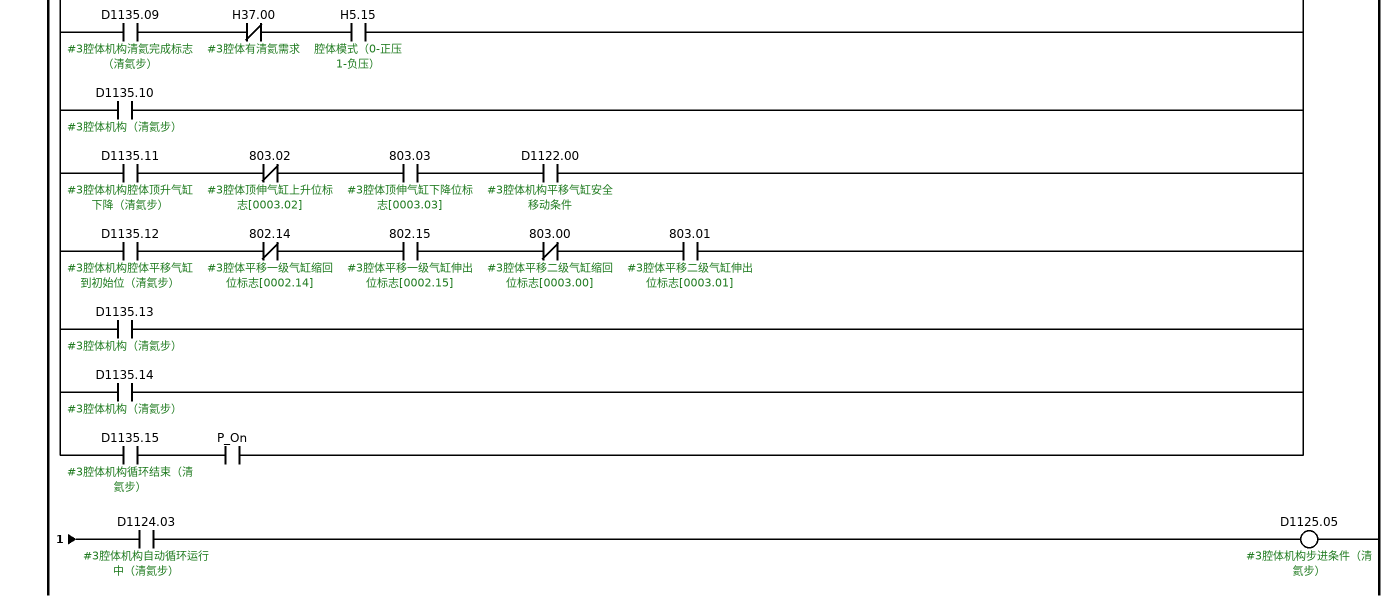
; [picture p312: 氦检机构 / 氦检腔3自动, rungs 23-23]
; rung 23
LD D1134.00  ; #3腔体机构自动开始（清氦步）
AND T1576  ; #3腔体机构开始运行延时（清氦步）
LD D1134.01  ; #3腔体机构平移气缸到氦检位/数据初始化（清氦步）
ANDNOT 802.14  ; #3腔体平移一级气缸缩回位标志[0002.14]
AND 802.15  ; #3腔体平移一级气缸伸出位标志[0002.15]
AND 803.00  ; #3腔体平移二级气缸缩回位标志[0003.00]
ANDNOT 803.01  ; #3腔体平移二级气缸伸出位标志[0003.01]
AND T2140  ; #3-1数据初始化延时（清氦）
ORLD
LD D1134.02  ; #3腔体机构腔体顶升气缸上升（清氦步）
AND 803.02  ; #3腔体顶伸气缸上升位标志[0003.02]
ANDNOT 803.03  ; #3腔体顶伸气缸下降位标志[0003.03]
ORLD
LD D1134.03  ; #3腔体机构氦检仪真空阀关闭（清氦步）
AND 820.11  ; 氦检仪真空阀关到位标志
ORLD
LD D1134.04  ; #3腔体机构正压开腔体阀/负压关腔体阀/氦检阀打开  // 负压模式下，复测前的清氦不允许抽电池
LDNOT H5.15  ; 腔体模式（0-正压 1-负压）
ORNOT D1127.01  ; #3腔体机构清氦需求判定（自动步）
LD 822.04  ; #3-1腔体阀开到位标志
AND 822.06  ; #3-2腔体阀开到位标志
LD D1130.11  ; #3腔体机构关闭#3-1腔体阀/清氦判定（自动单检步）
AND 822.04  ; #3-1腔体阀开到位标志
ORLD
LD D1131.07  ; #3腔体机构清氦需求判定（自动单检步）
AND 822.06  ; #3-2腔体阀开到位标志
ORLD
ANDLD
LD H5.15  ; 腔体模式（0-正压 1-负压）
AND D1127.01  ; #3腔体机构清氦需求判定（自动步）
AND 822.05  ; #3-1腔体阀关到位标志
AND 822.07  ; #3-2腔体阀关到位标志
ORLD
ANDLD
AND D1122.15  ; #3腔体机构腔体抽气阀打开允许
AND D1122.14  ; #3腔体氦检阀打开允许条件
AND 803.04  ; #3腔体氦检阀开到位标志[0003.04]
LD W380.15  ; 氦检仪漏率低于设定值（稳态）
OR H5.02  ; 氦检仪屏蔽
ANDLD
ORLD
OR D1134.05  ; #3腔体机构（清氦步）
LD D1134.06  ; #3腔体机构腔体抽气阀打开/电池抽气阀打开（清氦步）
LD T2100  ; #3-1腔体抽真空阈值到达延时（测试）
OR T2108  ; #3-1腔体抽残气时间上限到达延时（测试）
ANDLD
LD 824.04  ; #3-1电池抽真空阀开到位标志
AND T2120  ; #3-1电池抽真空阈值到达延时（测试）
OR T2121  ; #3-1电池抽真空时间上限到达延时（测试）
LD 824.06  ; #3-2电池抽真空阀开到位标志
AND T2420  ; #3-2电池抽真空阈值到达延时（测试）
OR T2421  ; #3-2电池抽真空时间上限到达延时（测试）
ANDLD
OR H5.15  ; 腔体模式（0-正压 1-负压）
OR H5.10  ; 空跑程序
ANDLD
ORLD
LD D1134.07  ; #3腔体机构腔体抽气阀关闭/电池抽气阀关闭（清氦步）
AND 822.03  ; #3腔体抽真空阀关到位标志
AND 824.05  ; #3-1电池抽真空阀关到位标志
AND 824.07  ; #3-2电池抽真空阀关到位标志
ORLD
OR D1134.08  ; #3腔体机构（清氦步）
LD D1134.09  ; #3腔体机构氦检清洁阀打开/电池破真空阀打开（清氦步）
AND T2141  ; #3-1清氦注氮时长（清氦）
LD T2122  ; #3-1电池破真空阈值到达延时（测试）
OR T2123  ; #3-1电池破真空时间上限到达延时（测试）
ANDLD
LD T2422  ; #3-2电池破真空阈值到达延时（测试）
OR T2423  ; #3-2电池破真空时间上限到达延时（测试）
ANDLD
ORLD
LD D1134.10  ; #3腔体机构氦检清洁阀关闭/电池破真空阀关闭（清氦步）
AND 820.13  ; 复检清洁阀关到位标志
AND 824.13  ; #3-1电池破真空阀关到位标志
AND 824.15  ; #3-2电池破真空阀关到位标志
ORLD
OR D1134.11  ; #3腔体机构（清氦步）
LD D1134.12  ; #3腔体机构清氦次数判定（清氦步）
AND>=(325) D472 D124  ; #3-1腔体管路清氦计数, 腔体测试设定清氦次数（次_UInt）
ORLD
OR D1134.13  ; #3腔体机构（清氦步）
LD D1134.14  ; #3腔体机构腔体抽气阀打开/电池抽气阀打开（清氦步）
AND 803.04  ; #3腔体氦检阀开到位标志[0003.04]
AND T2100  ; #3-1腔体抽真空阈值到达延时（测试）
LD 824.04  ; #3-1电池抽真空阀开到位标志
AND T2120  ; #3-1电池抽真空阈值到达延时（测试）
AND 824.06  ; #3-2电池抽真空阀开到位标志
AND T2420  ; #3-2电池抽真空阈值到达延时（测试）
OR H5.15  ; 腔体模式（0-正压 1-负压）
OR H5.10  ; 空跑程序
ANDLD
ORLD
LD D1134.15  ; #3腔体机构关闭电池抽气阀（清氦步）
AND 824.05  ; #3-1电池抽真空阀关到位标志
AND 824.07  ; #3-2电池抽真空阀关到位标志
ORLD
LD D1135.00  ; #3腔体机构腔体氦检阀仪真空阀打开/延时关腔体抽气阀（清氦步）
AND 803.04  ; #3腔体氦检阀开到位标志[0003.04]
AND 820.10  ; 氦检仪真空阀开到位标志
AND T2106  ; #3-1腔体氦检数据取值判定延时（测试）
ORLD
OR D1135.01  ; #3腔体机构（清氦步）
LD D1135.02  ; #3腔体机构腔体氦检阀关闭（清氦步）
AND 803.05  ; #3腔体氦检阀关到位标志[0003.05]
ORLD
LD D1135.03  ; #3腔体机构腔体抽气阀关闭/电池抽气阀关闭（清氦步）
AND 824.05  ; #3-1电池抽真空阀关到位标志
AND 824.07  ; #3-2电池抽真空阀关到位标志
AND 822.03  ; #3腔体抽真空阀关到位标志
ORLD
LD D1135.04  ; #3腔体机构是否需要重新清氦判定（清氦步）
ANDNOT H37.10  ; #3-1腔体清氦失败，重新进行清氦流程  // 清氦失败，重新进行清氦
ORLD
OR D1135.05  ; #3腔体机构（清氦步）
LD D1135.06  ; #3腔体机构开腔体破真空阀/开电池破真空阀/开腔体阀（清氦步）
AND T2102  ; #3-1腔体破真空阈值到达延时（测试）
AND T2122  ; #3-1电池破真空阈值到达延时（测试）
AND T2422  ; #3-2电池破真空阈值到达延时（测试）
ORLD
LD D1135.07  ; #3腔体机构关腔体破真空阀/关电池破真空阀（清氦步）
AND 822.09  ; #3腔体破真空阀关到位标志
AND 824.13  ; #3-1电池破真空阀关到位标志
AND 824.15  ; #3-2电池破真空阀关到位标志
ORLD
OR D1135.08  ; #3腔体机构（清氦步）
LD D1135.09  ; #3腔体机构清氦完成标志（清氦步）  // 正压腔体是待料清氦，需跳转回测试步序
ANDNOT H37.00  ; #3腔体有清氦需求
AND H5.15  ; 腔体模式（0-正压 1-负压）
ORLD
OR D1135.10  ; #3腔体机构（清氦步）
LD D1135.11  ; #3腔体机构腔体顶升气缸下降（清氦步）
ANDNOT 803.02  ; #3腔体顶伸气缸上升位标志[0003.02]
AND 803.03  ; #3腔体顶伸气缸下降位标志[0003.03]
AND D1122.00  ; #3腔体机构平移气缸安全移动条件
ORLD
LD D1135.12  ; #3腔体机构腔体平移气缸到初始位（清氦步）
ANDNOT 802.14  ; #3腔体平移一级气缸缩回位标志[0002.14]
AND 802.15  ; #3腔体平移一级气缸伸出位标志[0002.15]
ANDNOT 803.00  ; #3腔体平移二级气缸缩回位标志[0003.00]
AND 803.01  ; #3腔体平移二级气缸伸出位标志[0003.01]
ORLD
OR D1135.13  ; #3腔体机构（清氦步）
OR D1135.14  ; #3腔体机构（清氦步）
LD D1135.15  ; #3腔体机构循环结束（清氦步）
AND P_On
ORLD
AND D1124.03  ; #3腔体机构自动循环运行中（清氦步）
OUT D1125.05  ; #3腔体机构步进条件（清氦步）

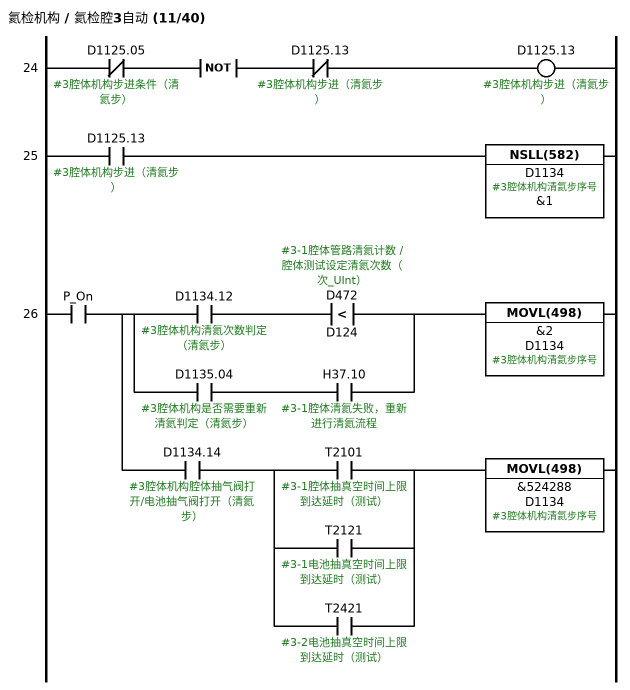
; rung 24
LDNOT D1125.05  ; #3腔体机构步进条件（清氦步）
NOT(520)
ANDNOT D1125.13  ; #3腔体机构步进（清氦步）
OUT D1125.13  ; #3腔体机构步进（清氦步）
; rung 25
LD D1125.13  ; #3腔体机构步进（清氦步）
NSLL(582) D1134 &1  ; #3腔体机构清氦步序号
; rung 26
LD P_On
OUT TR0
LD D1134.12  ; #3腔体机构清氦次数判定（清氦步）
AND<(310) D472 D124  ; #3-1腔体管路清氦计数, 腔体测试设定清氦次数（次_UInt）
LD D1135.04  ; #3腔体机构是否需要重新清氦判定（清氦步）
AND H37.10  ; #3-1腔体清氦失败，重新进行清氦流程  // 清氦失败，重新进行清氦
ORLD
ANDLD
MOVL(498) &2 D1134  ; #3腔体机构清氦步序号
LD TR0
AND D1134.14  ; #3腔体机构腔体抽气阀打开/电池抽气阀打开（清氦步）
LD T2101  ; #3-1腔体抽真空时间上限到达延时（测试）
OR T2121  ; #3-1电池抽真空时间上限到达延时（测试）
OR T2421  ; #3-2电池抽真空时间上限到达延时（测试）
ANDLD
MOVL(498) &524288 D1134  ; #3腔体机构清氦步序号  // 清氦过程腔体或电池抽气上限达到，均直接判定清氦完成，不进入氦检步序（跳转至D1075.03）

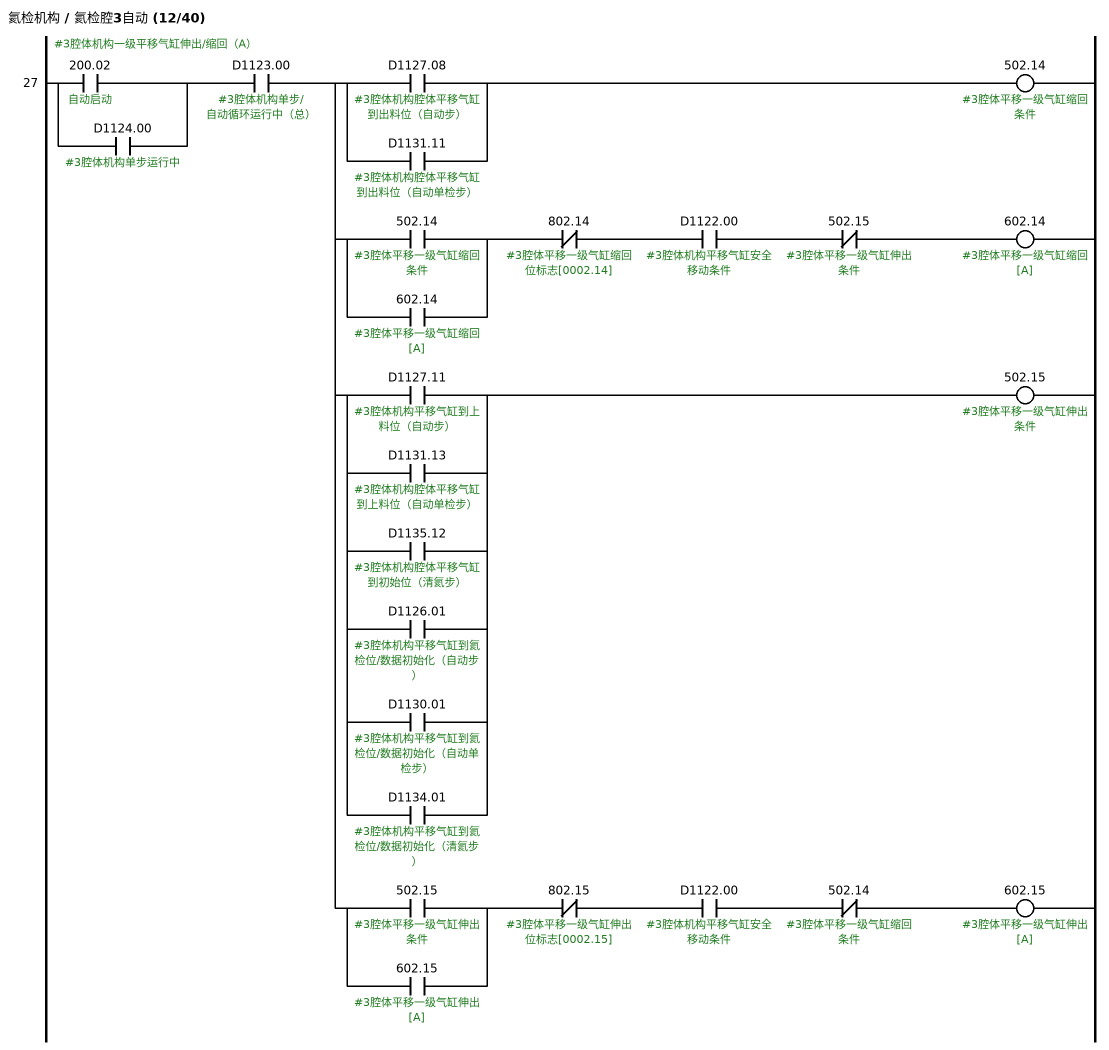
; rung 27: #3腔体机构一级平移气缸伸出/缩回（A）
LD 200.02  ; 自动启动
OR D1124.00  ; #3腔体机构单步运行中
AND D1123.00  ; #3腔体机构单步/自动循环运行中（总）
OUT TR0
LD D1127.08  ; #3腔体机构腔体平移气缸到出料位（自动步）
OR D1131.11  ; #3腔体机构腔体平移气缸到出料位（自动单检步）
ANDLD
OUT 502.14  ; #3腔体平移一级气缸缩回条件
LD TR0
LD 502.14  ; #3腔体平移一级气缸缩回条件
OR 602.14  ; #3腔体平移一级气缸缩回[A]
ANDLD
ANDNOT 802.14  ; #3腔体平移一级气缸缩回位标志[0002.14]
AND D1122.00  ; #3腔体机构平移气缸安全移动条件
ANDNOT 502.15  ; #3腔体平移一级气缸伸出条件
OUT 602.14  ; #3腔体平移一级气缸缩回[A]
LD TR0
LD D1127.11  ; #3腔体机构平移气缸到上料位（自动步）
OR D1131.13  ; #3腔体机构腔体平移气缸到上料位（自动单检步）
OR D1135.12  ; #3腔体机构腔体平移气缸到初始位（清氦步）
OR D1126.01  ; #3腔体机构平移气缸到氦检位/数据初始化（自动步）
OR D1130.01  ; #3腔体机构平移气缸到氦检位/数据初始化（自动单检步）
OR D1134.01  ; #3腔体机构平移气缸到氦检位/数据初始化（清氦步）
ANDLD
OUT 502.15  ; #3腔体平移一级气缸伸出条件
LD TR0
LD 502.15  ; #3腔体平移一级气缸伸出条件
OR 602.15  ; #3腔体平移一级气缸伸出[A]
ANDLD
ANDNOT 802.15  ; #3腔体平移一级气缸伸出位标志[0002.15]
AND D1122.00  ; #3腔体机构平移气缸安全移动条件
ANDNOT 502.14  ; #3腔体平移一级气缸缩回条件
OUT 602.15  ; #3腔体平移一级气缸伸出[A]

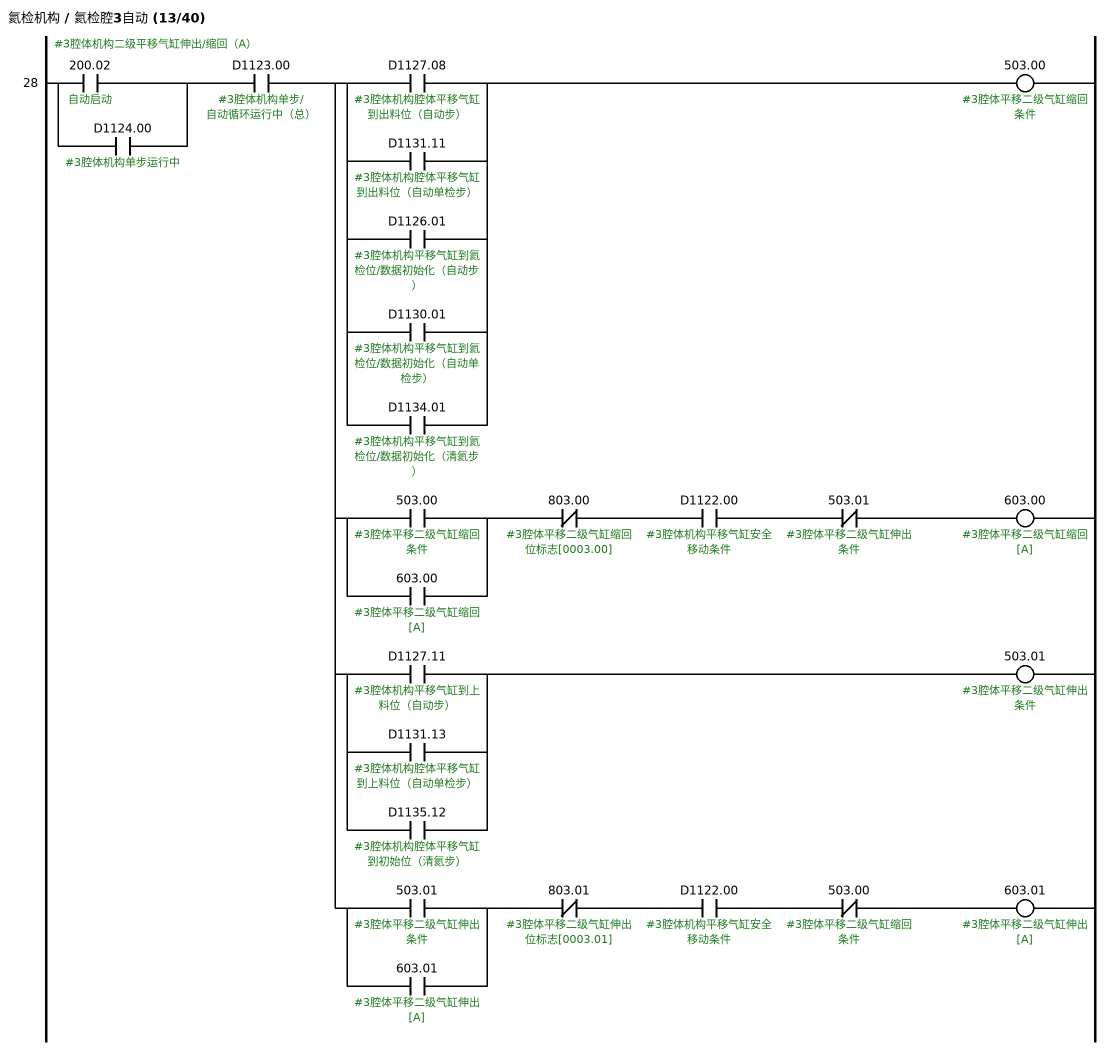
; rung 28: #3腔体机构二级平移气缸伸出/缩回（A）
LD 200.02  ; 自动启动
OR D1124.00  ; #3腔体机构单步运行中
AND D1123.00  ; #3腔体机构单步/自动循环运行中（总）
OUT TR0
LD D1127.08  ; #3腔体机构腔体平移气缸到出料位（自动步）
OR D1131.11  ; #3腔体机构腔体平移气缸到出料位（自动单检步）
OR D1126.01  ; #3腔体机构平移气缸到氦检位/数据初始化（自动步）
OR D1130.01  ; #3腔体机构平移气缸到氦检位/数据初始化（自动单检步）
OR D1134.01  ; #3腔体机构平移气缸到氦检位/数据初始化（清氦步）
ANDLD
OUT 503.00  ; #3腔体平移二级气缸缩回条件
LD TR0
LD 503.00  ; #3腔体平移二级气缸缩回条件
OR 603.00  ; #3腔体平移二级气缸缩回[A]
ANDLD
ANDNOT 803.00  ; #3腔体平移二级气缸缩回位标志[0003.00]
AND D1122.00  ; #3腔体机构平移气缸安全移动条件
ANDNOT 503.01  ; #3腔体平移二级气缸伸出条件
OUT 603.00  ; #3腔体平移二级气缸缩回[A]
LD TR0
LD D1127.11  ; #3腔体机构平移气缸到上料位（自动步）
OR D1131.13  ; #3腔体机构腔体平移气缸到上料位（自动单检步）
OR D1135.12  ; #3腔体机构腔体平移气缸到初始位（清氦步）
ANDLD
OUT 503.01  ; #3腔体平移二级气缸伸出条件
LD TR0
LD 503.01  ; #3腔体平移二级气缸伸出条件
OR 603.01  ; #3腔体平移二级气缸伸出[A]
ANDLD
ANDNOT 803.01  ; #3腔体平移二级气缸伸出位标志[0003.01]
AND D1122.00  ; #3腔体机构平移气缸安全移动条件
ANDNOT 503.00  ; #3腔体平移二级气缸缩回条件
OUT 603.01  ; #3腔体平移二级气缸伸出[A]

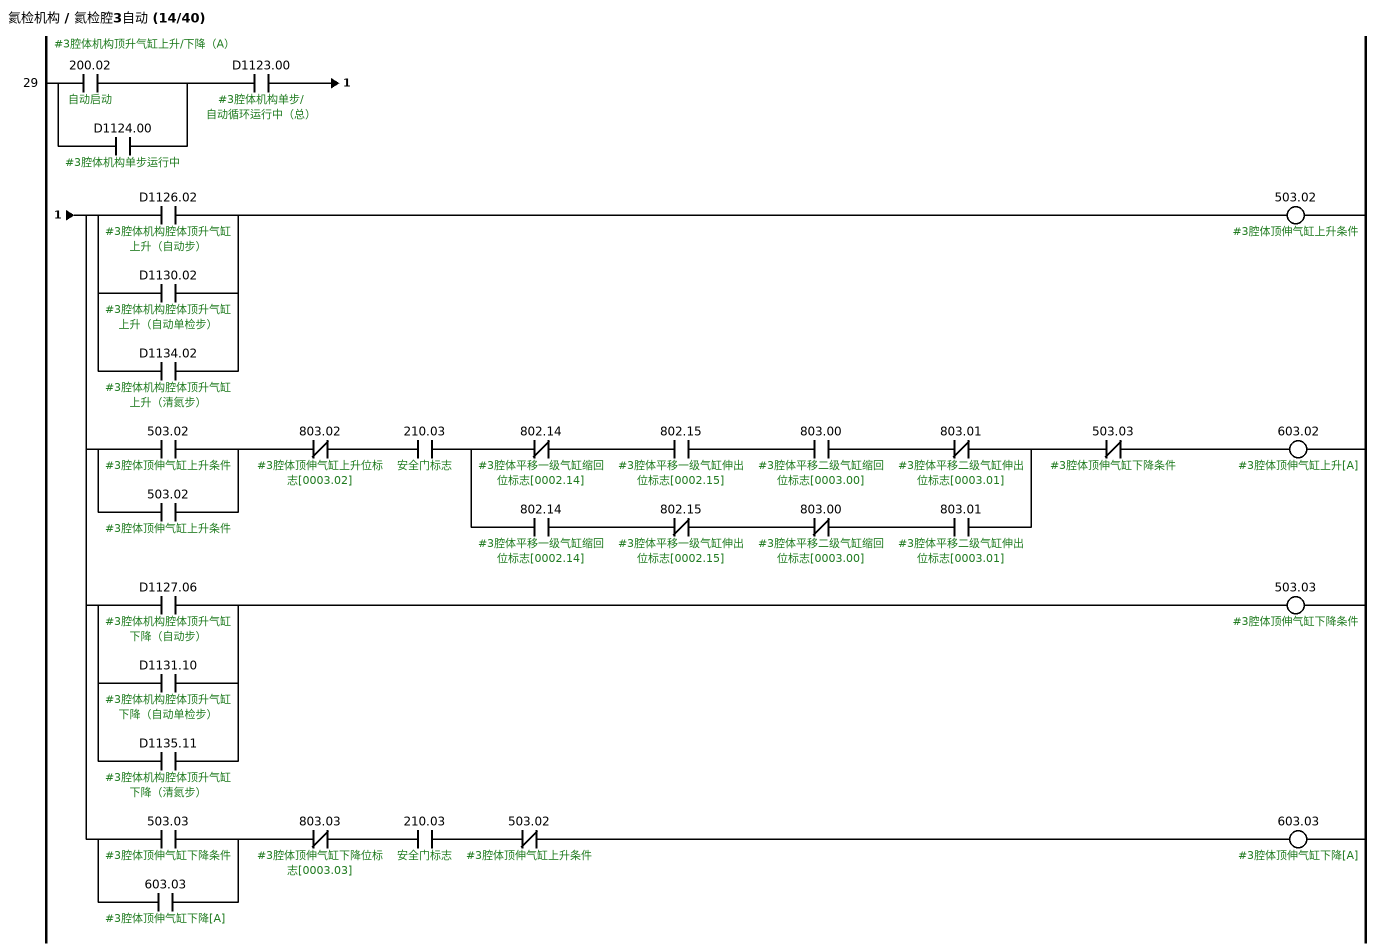
; rung 29: #3腔体机构顶升气缸上升/下降（A）
LD 200.02  ; 自动启动
OR D1124.00  ; #3腔体机构单步运行中
AND D1123.00  ; #3腔体机构单步/自动循环运行中（总）
OUT TR0
LD D1126.02  ; #3腔体机构腔体顶升气缸上升（自动步）
OR D1130.02  ; #3腔体机构腔体顶升气缸上升（自动单检步）
OR D1134.02  ; #3腔体机构腔体顶升气缸上升（清氦步）
ANDLD
OUT 503.02  ; #3腔体顶伸气缸上升条件
LD TR0
LD 503.02  ; #3腔体顶伸气缸上升条件
OR 503.02  ; #3腔体顶伸气缸上升条件
ANDLD
ANDNOT 803.02  ; #3腔体顶伸气缸上升位标志[0003.02]
AND 210.03  ; 安全门标志
LDNOT 802.14  ; #3腔体平移一级气缸缩回位标志[0002.14]
AND 802.15  ; #3腔体平移一级气缸伸出位标志[0002.15]
AND 803.00  ; #3腔体平移二级气缸缩回位标志[0003.00]
ANDNOT 803.01  ; #3腔体平移二级气缸伸出位标志[0003.01]
LD 802.14  ; #3腔体平移一级气缸缩回位标志[0002.14]
ANDNOT 802.15  ; #3腔体平移一级气缸伸出位标志[0002.15]
ANDNOT 803.00  ; #3腔体平移二级气缸缩回位标志[0003.00]
AND 803.01  ; #3腔体平移二级气缸伸出位标志[0003.01]
ORLD
ANDLD
ANDNOT 503.03  ; #3腔体顶伸气缸下降条件
OUT 603.02  ; #3腔体顶伸气缸上升[A]
LD TR0
LD D1127.06  ; #3腔体机构腔体顶升气缸下降（自动步）
OR D1131.10  ; #3腔体机构腔体顶升气缸下降（自动单检步）
OR D1135.11  ; #3腔体机构腔体顶升气缸下降（清氦步）
ANDLD
OUT 503.03  ; #3腔体顶伸气缸下降条件
LD TR0
LD 503.03  ; #3腔体顶伸气缸下降条件
OR 603.03  ; #3腔体顶伸气缸下降[A]
ANDLD
ANDNOT 803.03  ; #3腔体顶伸气缸下降位标志[0003.03]
AND 210.03  ; 安全门标志
ANDNOT 503.02  ; #3腔体顶伸气缸上升条件
OUT 603.03  ; #3腔体顶伸气缸下降[A]

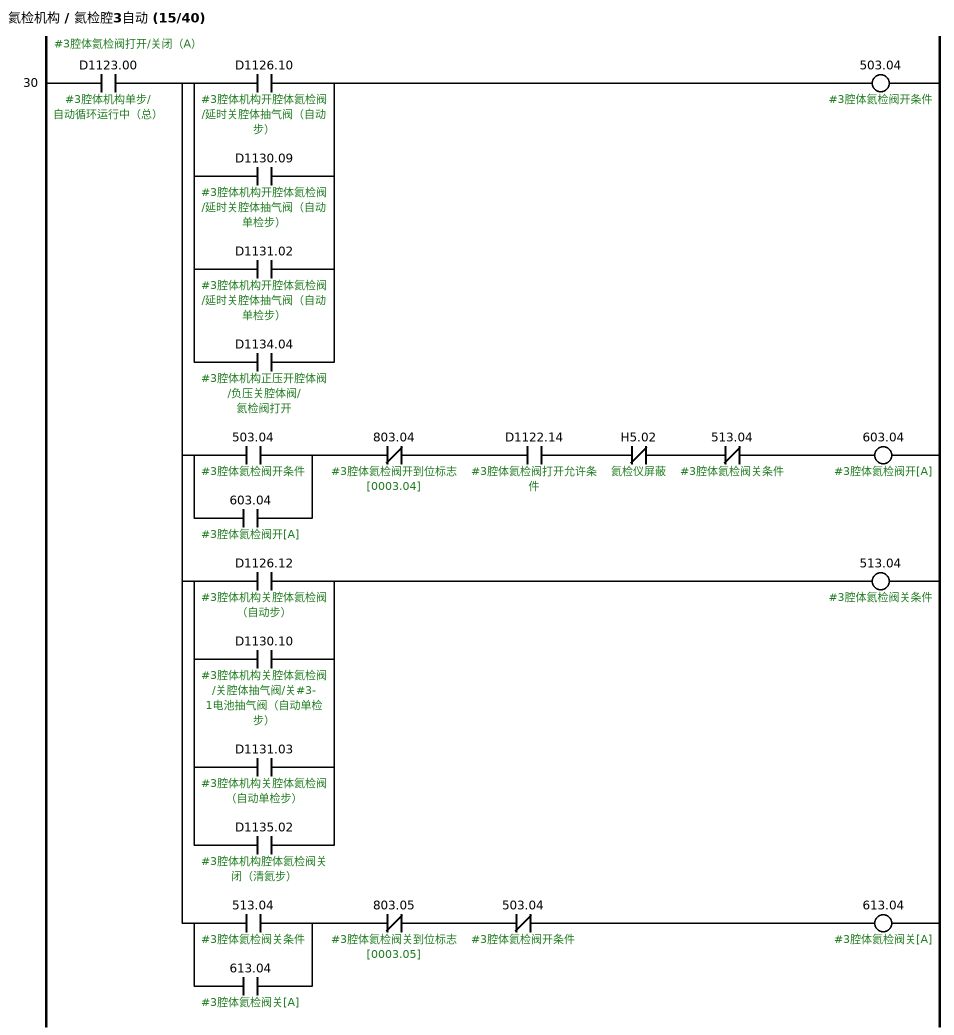
; rung 30: #3腔体氦检阀打开/关闭（A）
LD D1123.00  ; #3腔体机构单步/自动循环运行中（总）
OUT TR0
LD D1126.10  ; #3腔体机构开腔体氦检阀/延时关腔体抽气阀（自动步）
OR D1130.09  ; #3腔体机构开腔体氦检阀/延时关腔体抽气阀（自动单检步）
OR D1131.02  ; #3腔体机构开腔体氦检阀/延时关腔体抽气阀（自动单检步）
OR D1134.04  ; #3腔体机构正压开腔体阀/负压关腔体阀/氦检阀打开
ANDLD
OUT 503.04  ; #3腔体氦检阀开条件
LD TR0
LD 503.04  ; #3腔体氦检阀开条件
OR 603.04  ; #3腔体氦检阀开[A]
ANDLD
ANDNOT 803.04  ; #3腔体氦检阀开到位标志[0003.04]
AND D1122.14  ; #3腔体氦检阀打开允许条件
ANDNOT H5.02  ; 氦检仪屏蔽
ANDNOT 513.04  ; #3腔体氦检阀关条件
OUT 603.04  ; #3腔体氦检阀开[A]
LD TR0
LD D1126.12  ; #3腔体机构关腔体氦检阀（自动步）
OR D1130.10  ; #3腔体机构关腔体氦检阀/关腔体抽气阀/关#3-1电池抽气阀（自动单检步）
OR D1131.03  ; #3腔体机构关腔体氦检阀（自动单检步）
OR D1135.02  ; #3腔体机构腔体氦检阀关闭（清氦步）
ANDLD
OUT 513.04  ; #3腔体氦检阀关条件
LD TR0
LD 513.04  ; #3腔体氦检阀关条件
OR 613.04  ; #3腔体氦检阀关[A]
ANDLD
ANDNOT 803.05  ; #3腔体氦检阀关到位标志[0003.05]
ANDNOT 503.04  ; #3腔体氦检阀开条件
OUT 613.04  ; #3腔体氦检阀关[A]

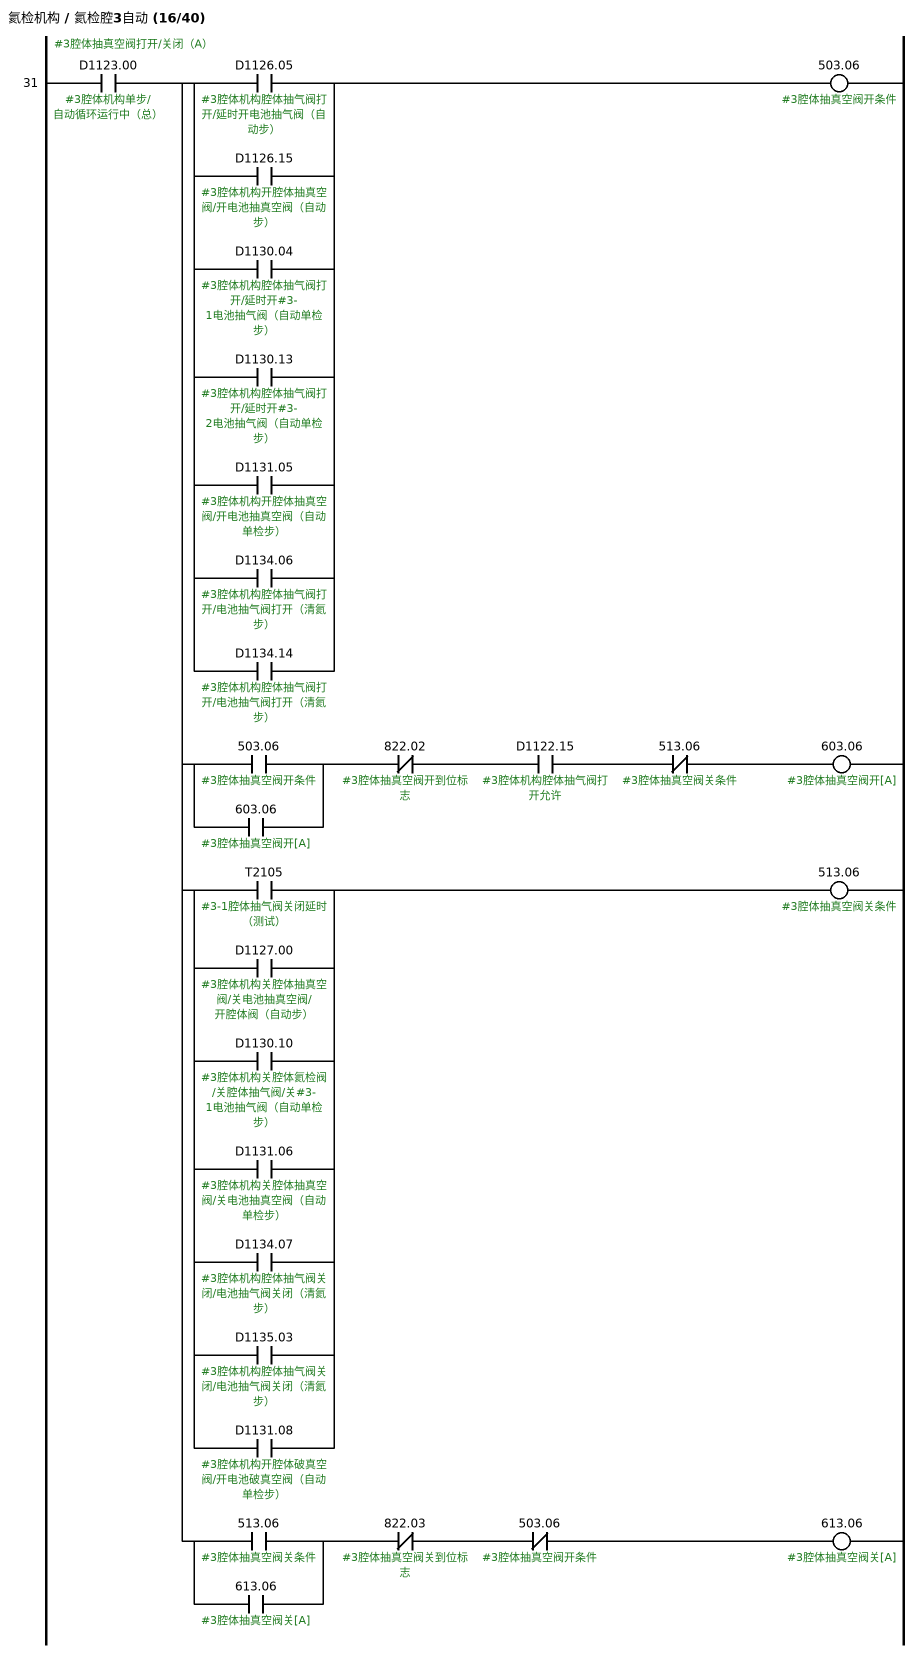
; rung 31: #3腔体抽真空阀打开/关闭（A）
LD D1123.00  ; #3腔体机构单步/自动循环运行中（总）
OUT TR0
LD D1126.05  ; #3腔体机构腔体抽气阀打开/延时开电池抽气阀（自动步）
OR D1126.15  ; #3腔体机构开腔体抽真空阀/开电池抽真空阀（自动步）
OR D1130.04  ; #3腔体机构腔体抽气阀打开/延时开#3-1电池抽气阀（自动单检步）
OR D1130.13  ; #3腔体机构腔体抽气阀打开/延时开#3-2电池抽气阀（自动单检步）
OR D1131.05  ; #3腔体机构开腔体抽真空阀/开电池抽真空阀（自动单检步）
OR D1134.06  ; #3腔体机构腔体抽气阀打开/电池抽气阀打开（清氦步）
OR D1134.14  ; #3腔体机构腔体抽气阀打开/电池抽气阀打开（清氦步）
ANDLD
OUT 503.06  ; #3腔体抽真空阀开条件
LD TR0
LD 503.06  ; #3腔体抽真空阀开条件
OR 603.06  ; #3腔体抽真空阀开[A]
ANDLD
ANDNOT 822.02  ; #3腔体抽真空阀开到位标志
AND D1122.15  ; #3腔体机构腔体抽气阀打开允许
ANDNOT 513.06  ; #3腔体抽真空阀关条件
OUT 603.06  ; #3腔体抽真空阀开[A]
LD TR0
LD T2105  ; #3-1腔体抽气阀关闭延时（测试）
OR D1127.00  ; #3腔体机构关腔体抽真空阀/关电池抽真空阀/开腔体阀（自动步）
OR D1130.10  ; #3腔体机构关腔体氦检阀/关腔体抽气阀/关#3-1电池抽气阀（自动单检步）
OR D1131.06  ; #3腔体机构关腔体抽真空阀/关电池抽真空阀（自动单检步）
OR D1134.07  ; #3腔体机构腔体抽气阀关闭/电池抽气阀关闭（清氦步）
OR D1135.03  ; #3腔体机构腔体抽气阀关闭/电池抽气阀关闭（清氦步）
OR D1131.08  ; #3腔体机构开腔体破真空阀/开电池破真空阀（自动单检步）
ANDLD
OUT 513.06  ; #3腔体抽真空阀关条件
LD TR0
LD 513.06  ; #3腔体抽真空阀关条件
OR 613.06  ; #3腔体抽真空阀关[A]
ANDLD
ANDNOT 822.03  ; #3腔体抽真空阀关到位标志
ANDNOT 503.06  ; #3腔体抽真空阀开条件
OUT 613.06  ; #3腔体抽真空阀关[A]

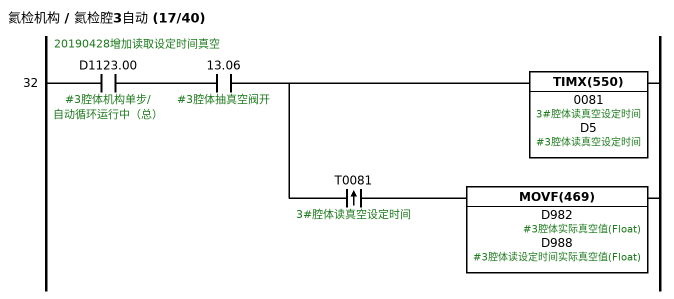
; rung 32: 20190428增加读取设定时间真空
LD D1123.00  ; #3腔体机构单步/自动循环运行中（总）
AND 13.06  ; #3腔体抽真空阀开
TIMX(550) 0081 D5  ; #3腔体读真空设定时间, 3#腔体读真空设定时间
@AND T0081  ; 3#腔体读真空设定时间
MOVF(469) D982 D988  ; #3腔体实际真空值(Float), #3腔体读设定时间实际真空值(Float)

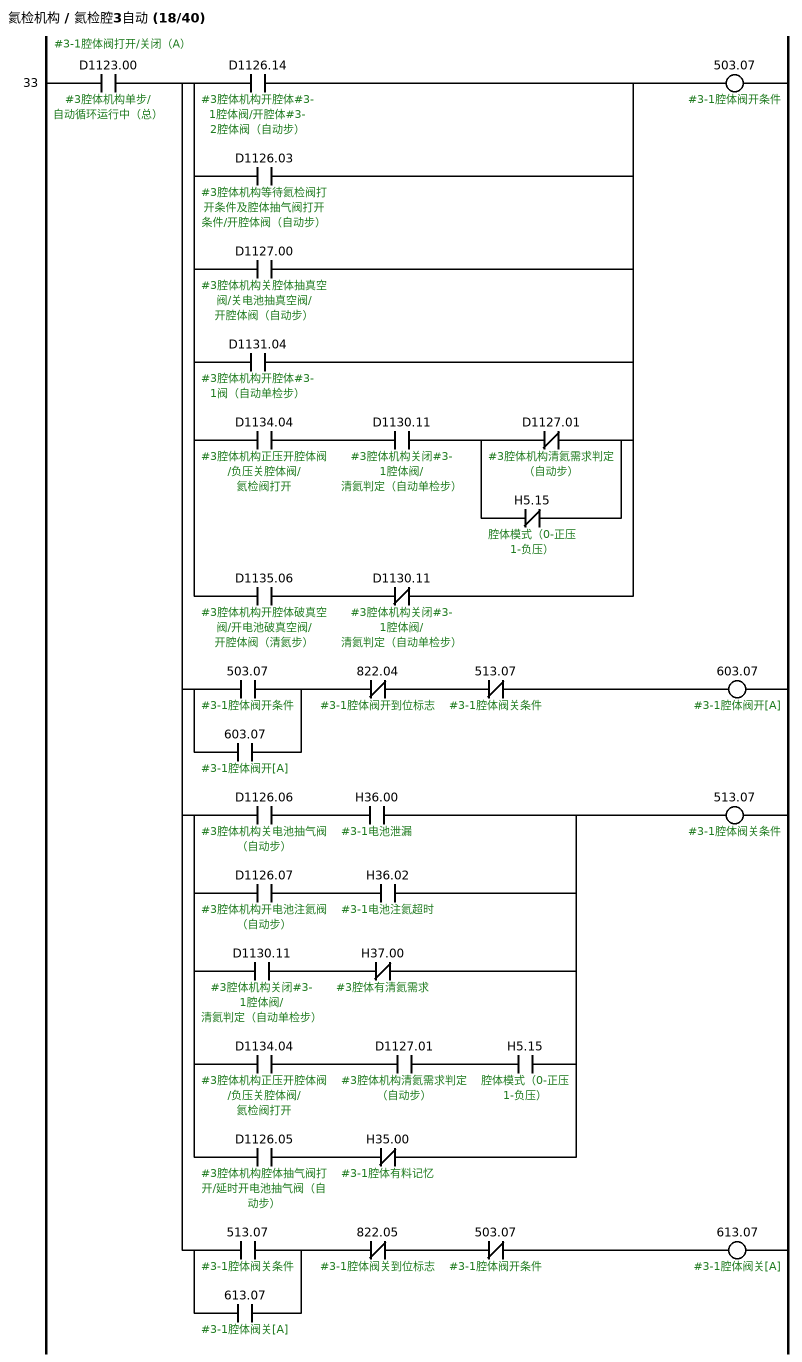
; rung 33: #3-1腔体阀打开/关闭（A）
LD D1123.00  ; #3腔体机构单步/自动循环运行中（总）
OUT TR0
LD D1126.14  ; #3腔体机构开腔体#3-1腔体阀/开腔体#3-2腔体阀（自动步）
OR D1126.03  ; #3腔体机构等待氦检阀打开条件及腔体抽气阀打开条件/开腔体阀（自动步）
OR D1127.00  ; #3腔体机构关腔体抽真空阀/关电池抽真空阀/开腔体阀（自动步）
OR D1131.04  ; #3腔体机构开腔体#3-1阀（自动单检步）
LD D1134.04  ; #3腔体机构正压开腔体阀/负压关腔体阀/氦检阀打开
AND D1130.11  ; #3腔体机构关闭#3-1腔体阀/清氦判定（自动单检步）
LDNOT D1127.01  ; #3腔体机构清氦需求判定（自动步）
ORNOT H5.15  ; 腔体模式（0-正压 1-负压）
ANDLD
ORLD
LD D1135.06  ; #3腔体机构开腔体破真空阀/开电池破真空阀/开腔体阀（清氦步）
ANDNOT D1130.11  ; #3腔体机构关闭#3-1腔体阀/清氦判定（自动单检步）
ORLD
ANDLD
OUT 503.07  ; #3-1腔体阀开条件
LD TR0
LD 503.07  ; #3-1腔体阀开条件
OR 603.07  ; #3-1腔体阀开[A]
ANDLD
ANDNOT 822.04  ; #3-1腔体阀开到位标志
ANDNOT 513.07  ; #3-1腔体阀关条件
OUT 603.07  ; #3-1腔体阀开[A]
LD TR0
LD D1126.06  ; #3腔体机构关电池抽气阀（自动步）
AND H36.00  ; #3-1电池泄漏
LD D1126.07  ; #3腔体机构开电池注氦阀（自动步）
AND H36.02  ; #3-1电池注氦超时
ORLD
LD D1130.11  ; #3腔体机构关闭#3-1腔体阀/清氦判定（自动单检步）
ANDNOT H37.00  ; #3腔体有清氦需求
ORLD
LD D1134.04  ; #3腔体机构正压开腔体阀/负压关腔体阀/氦检阀打开
AND D1127.01  ; #3腔体机构清氦需求判定（自动步）
AND H5.15  ; 腔体模式（0-正压 1-负压）
ORLD
LD D1126.05  ; #3腔体机构腔体抽气阀打开/延时开电池抽气阀（自动步）  // #1-1无料时不测试
ANDNOT H35.00  ; #3-1腔体有料记忆
ORLD
ANDLD
OUT 513.07  ; #3-1腔体阀关条件
LD TR0
LD 513.07  ; #3-1腔体阀关条件
OR 613.07  ; #3-1腔体阀关[A]
ANDLD
ANDNOT 822.05  ; #3-1腔体阀关到位标志
ANDNOT 503.07  ; #3-1腔体阀开条件
OUT 613.07  ; #3-1腔体阀关[A]

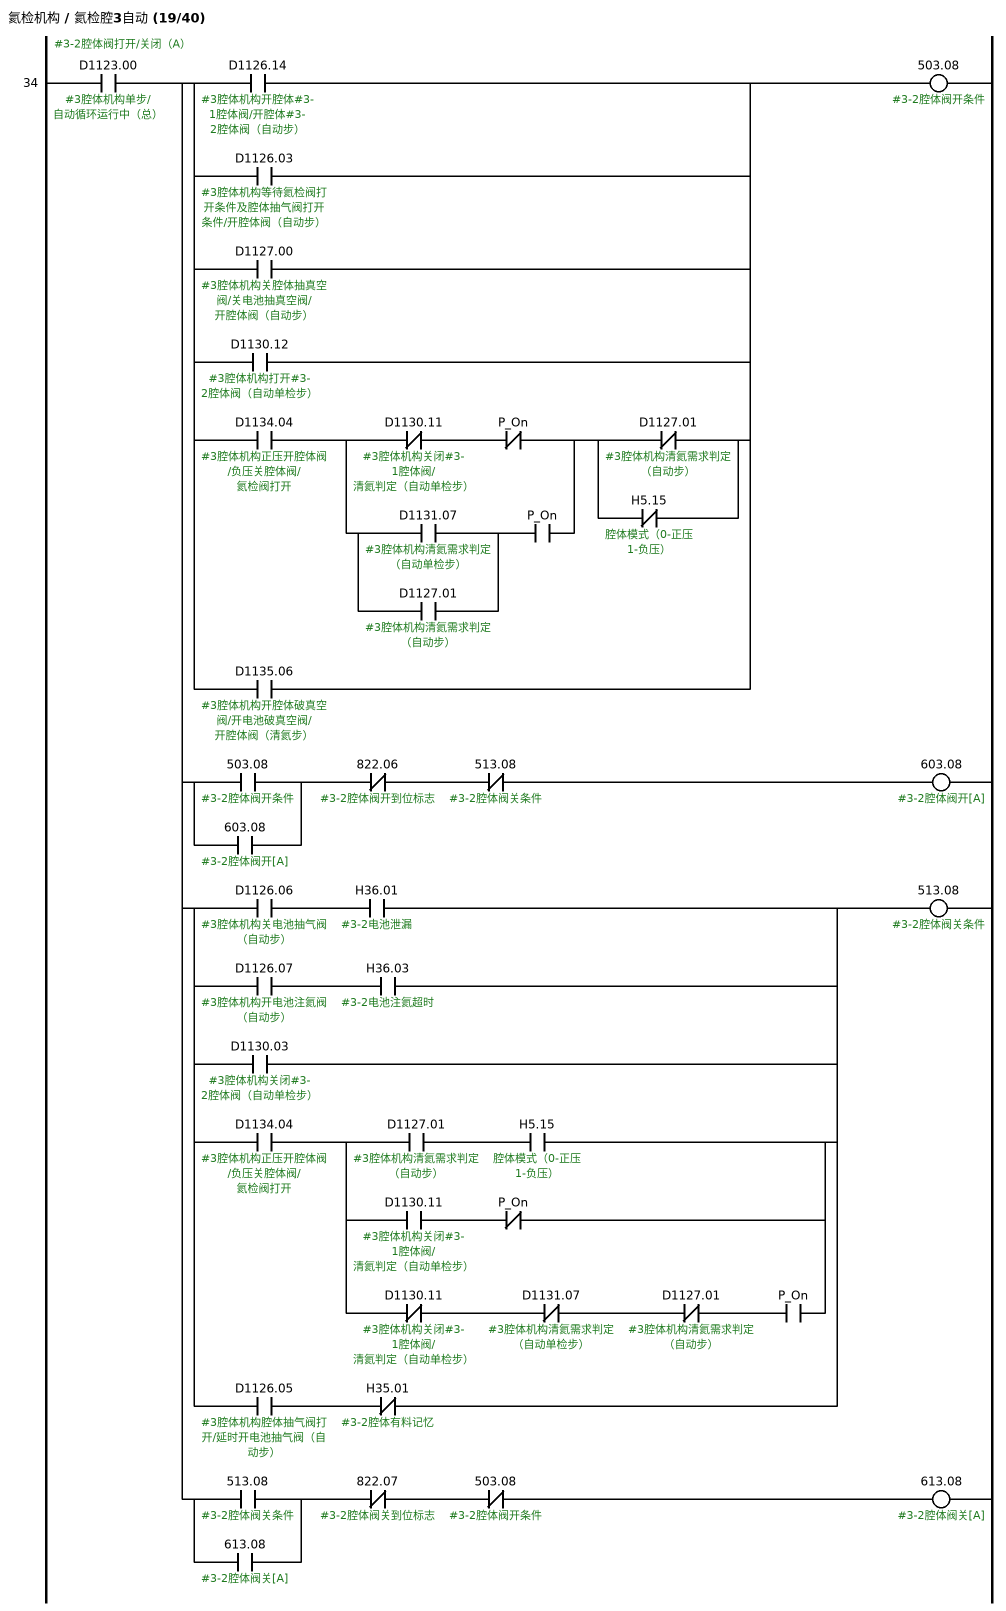
; rung 34: #3-2腔体阀打开/关闭（A）
LD D1123.00  ; #3腔体机构单步/自动循环运行中（总）
OUT TR0
LD D1126.14  ; #3腔体机构开腔体#3-1腔体阀/开腔体#3-2腔体阀（自动步）
OR D1126.03  ; #3腔体机构等待氦检阀打开条件及腔体抽气阀打开条件/开腔体阀（自动步）
OR D1127.00  ; #3腔体机构关腔体抽真空阀/关电池抽真空阀/开腔体阀（自动步）
OR D1130.12  ; #3腔体机构打开#3-2腔体阀（自动单检步）
LD D1134.04  ; #3腔体机构正压开腔体阀/负压关腔体阀/氦检阀打开
LDNOT D1130.11  ; #3腔体机构关闭#3-1腔体阀/清氦判定（自动单检步）
ANDNOT P_On
LD D1131.07  ; #3腔体机构清氦需求判定（自动单检步）
OR D1127.01  ; #3腔体机构清氦需求判定（自动步）
AND P_On
ORLD
ANDLD
LDNOT D1127.01  ; #3腔体机构清氦需求判定（自动步）
ORNOT H5.15  ; 腔体模式（0-正压 1-负压）
ANDLD
ORLD
OR D1135.06  ; #3腔体机构开腔体破真空阀/开电池破真空阀/开腔体阀（清氦步）
ANDLD
OUT 503.08  ; #3-2腔体阀开条件
LD TR0
LD 503.08  ; #3-2腔体阀开条件
OR 603.08  ; #3-2腔体阀开[A]
ANDLD
ANDNOT 822.06  ; #3-2腔体阀开到位标志
ANDNOT 513.08  ; #3-2腔体阀关条件
OUT 603.08  ; #3-2腔体阀开[A]
LD TR0
LD D1126.06  ; #3腔体机构关电池抽气阀（自动步）
AND H36.01  ; #3-2电池泄漏
LD D1126.07  ; #3腔体机构开电池注氦阀（自动步）
AND H36.03  ; #3-2电池注氦超时
ORLD
OR D1130.03  ; #3腔体机构关闭#3-2腔体阀（自动单检步）
LD D1134.04  ; #3腔体机构正压开腔体阀/负压关腔体阀/氦检阀打开
LD D1127.01  ; #3腔体机构清氦需求判定（自动步）
AND H5.15  ; 腔体模式（0-正压 1-负压）
LD D1130.11  ; #3腔体机构关闭#3-1腔体阀/清氦判定（自动单检步）
ANDNOT P_On
ORLD
LDNOT D1130.11  ; #3腔体机构关闭#3-1腔体阀/清氦判定（自动单检步）
ANDNOT D1131.07  ; #3腔体机构清氦需求判定（自动单检步）
ANDNOT D1127.01  ; #3腔体机构清氦需求判定（自动步）
AND P_On
ORLD
ANDLD
ORLD
LD D1126.05  ; #3腔体机构腔体抽气阀打开/延时开电池抽气阀（自动步）  // #1-2无料时不测试
ANDNOT H35.01  ; #3-2腔体有料记忆
ORLD
ANDLD
OUT 513.08  ; #3-2腔体阀关条件
LD TR0
LD 513.08  ; #3-2腔体阀关条件
OR 613.08  ; #3-2腔体阀关[A]
ANDLD
ANDNOT 822.07  ; #3-2腔体阀关到位标志
ANDNOT 503.08  ; #3-2腔体阀开条件
OUT 613.08  ; #3-2腔体阀关[A]

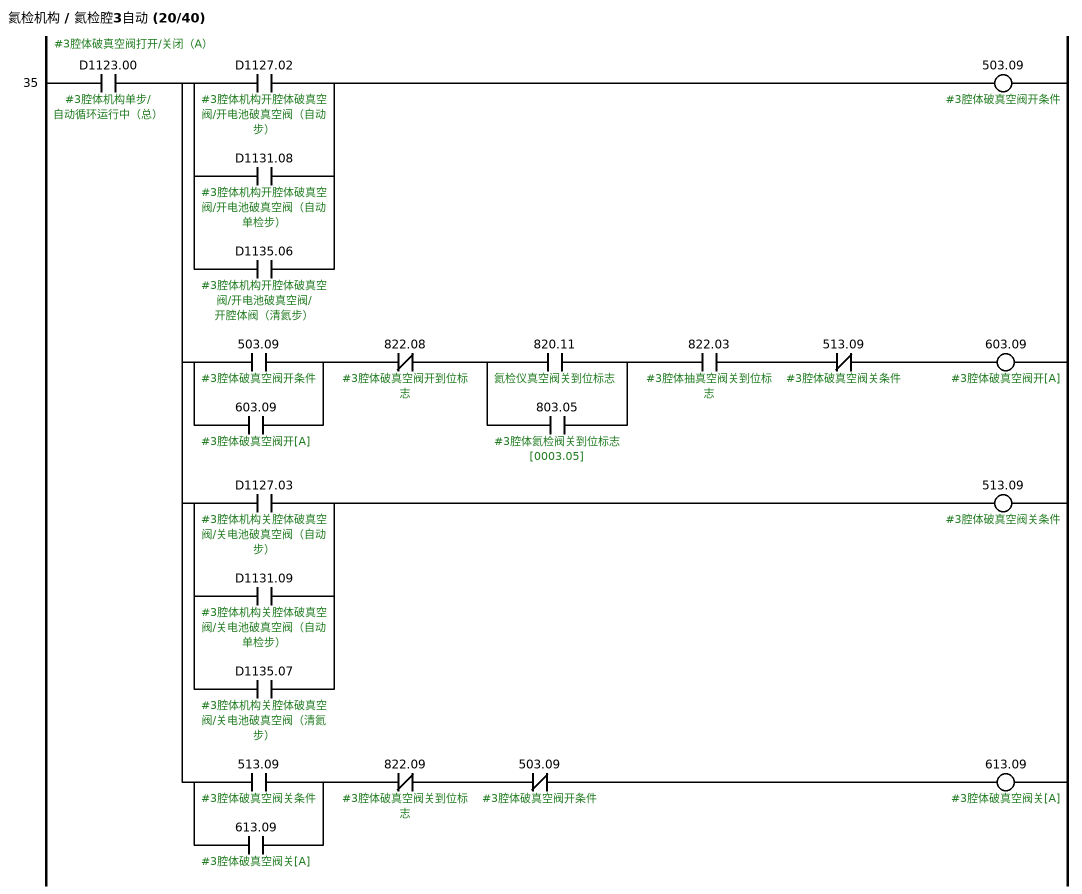
; rung 35: #3腔体破真空阀打开/关闭（A）
LD D1123.00  ; #3腔体机构单步/自动循环运行中（总）
OUT TR0
LD D1127.02  ; #3腔体机构开腔体破真空阀/开电池破真空阀（自动步）
OR D1131.08  ; #3腔体机构开腔体破真空阀/开电池破真空阀（自动单检步）
OR D1135.06  ; #3腔体机构开腔体破真空阀/开电池破真空阀/开腔体阀（清氦步）
ANDLD
OUT 503.09  ; #3腔体破真空阀开条件
LD TR0
LD 503.09  ; #3腔体破真空阀开条件
OR 603.09  ; #3腔体破真空阀开[A]
ANDLD
ANDNOT 822.08  ; #3腔体破真空阀开到位标志
LD 820.11  ; 氦检仪真空阀关到位标志
OR 803.05  ; #3腔体氦检阀关到位标志[0003.05]
ANDLD
AND 822.03  ; #3腔体抽真空阀关到位标志
ANDNOT 513.09  ; #3腔体破真空阀关条件
OUT 603.09  ; #3腔体破真空阀开[A]
LD TR0
LD D1127.03  ; #3腔体机构关腔体破真空阀/关电池破真空阀（自动步）
OR D1131.09  ; #3腔体机构关腔体破真空阀/关电池破真空阀（自动单检步）
OR D1135.07  ; #3腔体机构关腔体破真空阀/关电池破真空阀（清氦步）
ANDLD
OUT 513.09  ; #3腔体破真空阀关条件
LD TR0
LD 513.09  ; #3腔体破真空阀关条件
OR 613.09  ; #3腔体破真空阀关[A]
ANDLD
ANDNOT 822.09  ; #3腔体破真空阀关到位标志
ANDNOT 503.09  ; #3腔体破真空阀开条件
OUT 613.09  ; #3腔体破真空阀关[A]

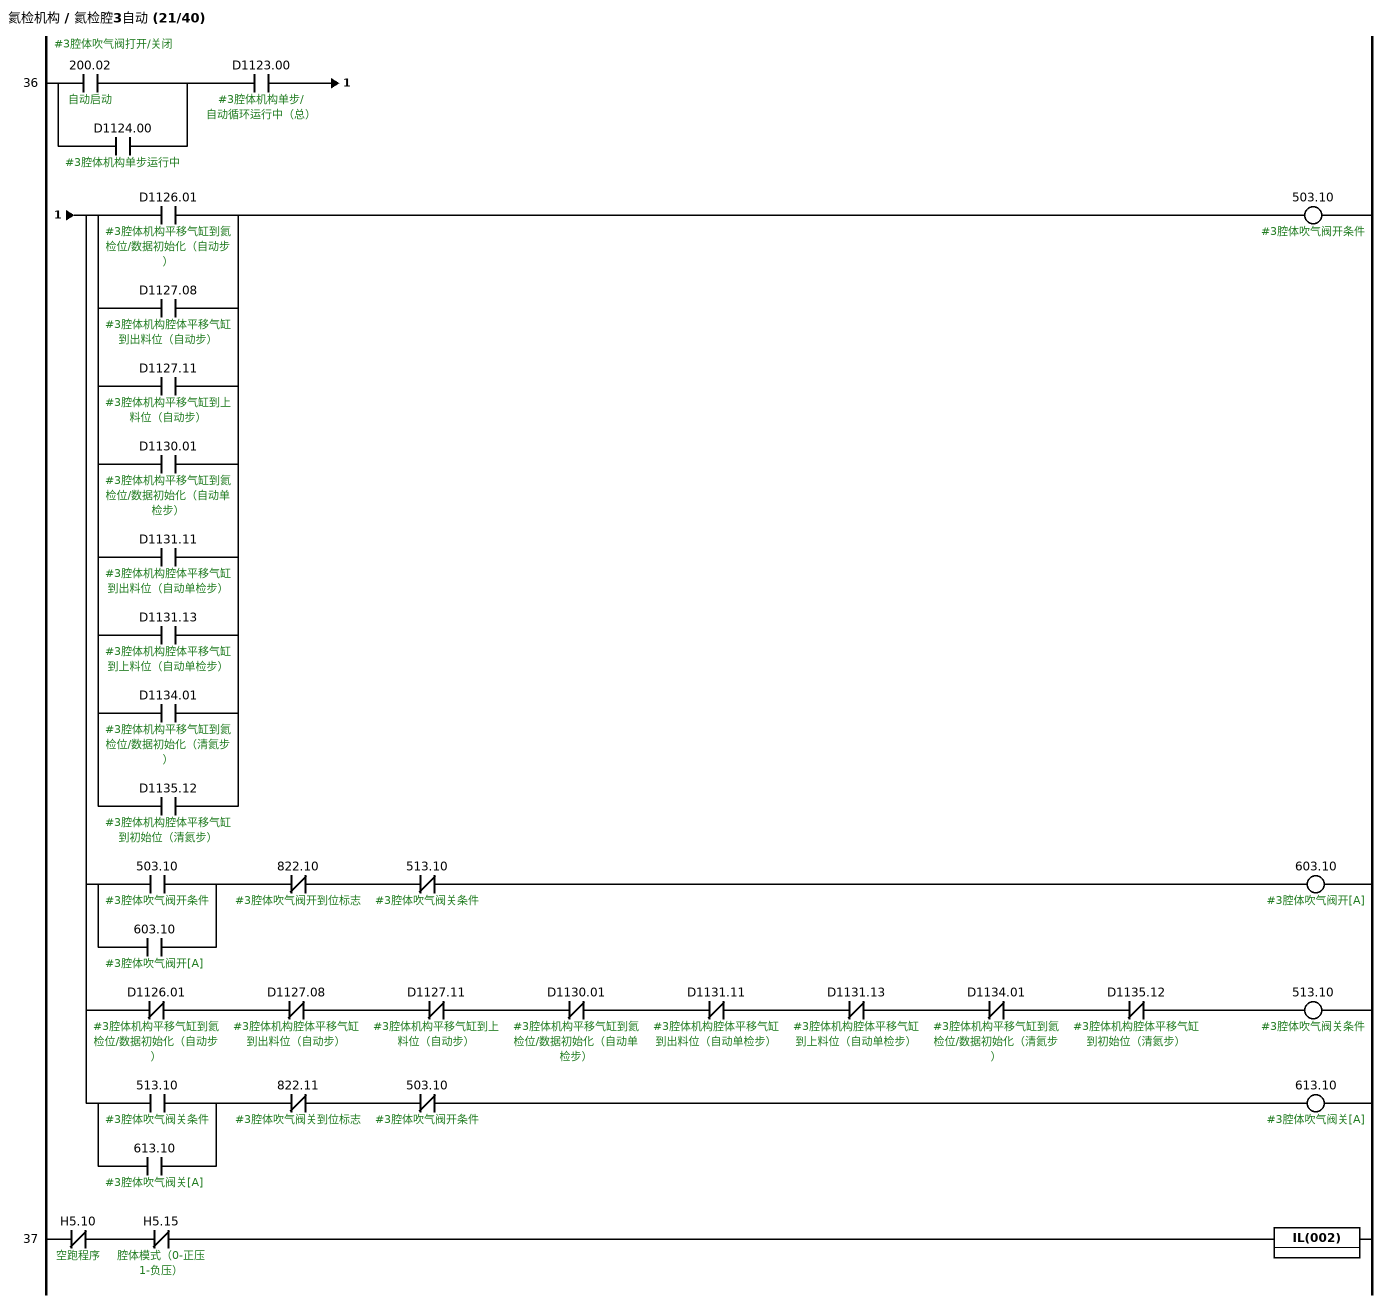
; rung 36: #3腔体吹气阀打开/关闭
LD 200.02  ; 自动启动
OR D1124.00  ; #3腔体机构单步运行中
AND D1123.00  ; #3腔体机构单步/自动循环运行中（总）
OUT TR0
LD D1126.01  ; #3腔体机构平移气缸到氦检位/数据初始化（自动步）
OR D1127.08  ; #3腔体机构腔体平移气缸到出料位（自动步）
OR D1127.11  ; #3腔体机构平移气缸到上料位（自动步）
OR D1130.01  ; #3腔体机构平移气缸到氦检位/数据初始化（自动单检步）
OR D1131.11  ; #3腔体机构腔体平移气缸到出料位（自动单检步）
OR D1131.13  ; #3腔体机构腔体平移气缸到上料位（自动单检步）
OR D1134.01  ; #3腔体机构平移气缸到氦检位/数据初始化（清氦步）
OR D1135.12  ; #3腔体机构腔体平移气缸到初始位（清氦步）
ANDLD
OUT 503.10  ; #3腔体吹气阀开条件
LD TR0
LD 503.10  ; #3腔体吹气阀开条件
OR 603.10  ; #3腔体吹气阀开[A]
ANDLD
ANDNOT 822.10  ; #3腔体吹气阀开到位标志
ANDNOT 513.10  ; #3腔体吹气阀关条件
OUT 603.10  ; #3腔体吹气阀开[A]
LD TR0
ANDNOT D1126.01  ; #3腔体机构平移气缸到氦检位/数据初始化（自动步）
ANDNOT D1127.08  ; #3腔体机构腔体平移气缸到出料位（自动步）
ANDNOT D1127.11  ; #3腔体机构平移气缸到上料位（自动步）
ANDNOT D1130.01  ; #3腔体机构平移气缸到氦检位/数据初始化（自动单检步）
ANDNOT D1131.11  ; #3腔体机构腔体平移气缸到出料位（自动单检步）
ANDNOT D1131.13  ; #3腔体机构腔体平移气缸到上料位（自动单检步）
ANDNOT D1134.01  ; #3腔体机构平移气缸到氦检位/数据初始化（清氦步）
ANDNOT D1135.12  ; #3腔体机构腔体平移气缸到初始位（清氦步）
OUT 513.10  ; #3腔体吹气阀关条件
LD TR0
LD 513.10  ; #3腔体吹气阀关条件
OR 613.10  ; #3腔体吹气阀关[A]
ANDLD
ANDNOT 822.11  ; #3腔体吹气阀关到位标志
ANDNOT 503.10  ; #3腔体吹气阀开条件
OUT 613.10  ; #3腔体吹气阀关[A]
; rung 37
LDNOT H5.10  ; 空跑程序
ANDNOT H5.15  ; 腔体模式（0-正压 1-负压）
IL(002)

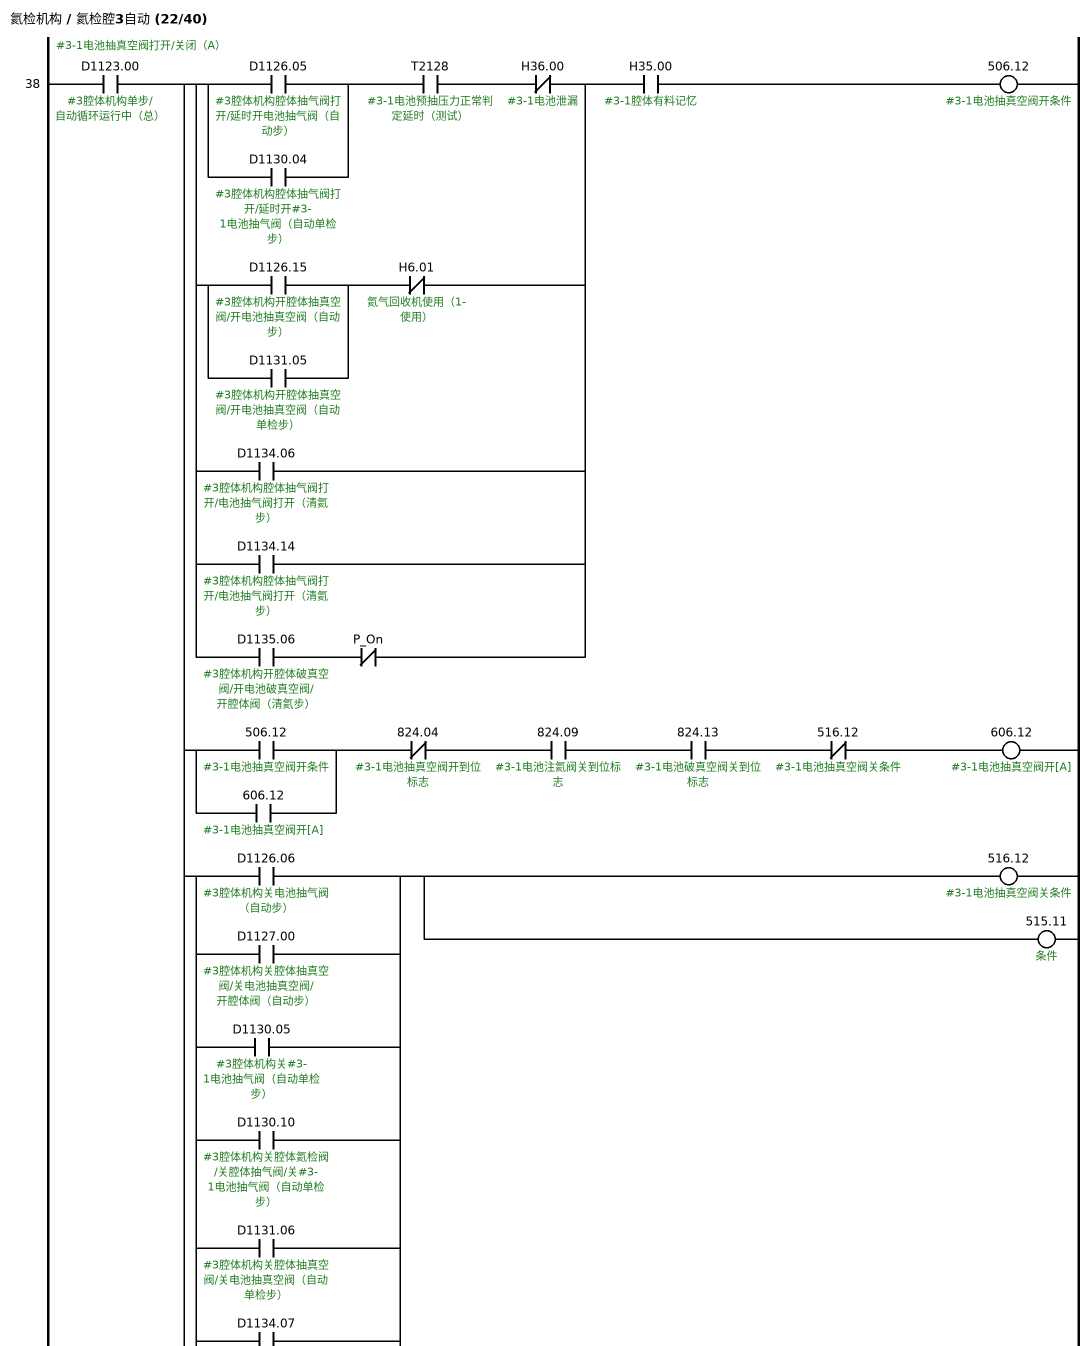

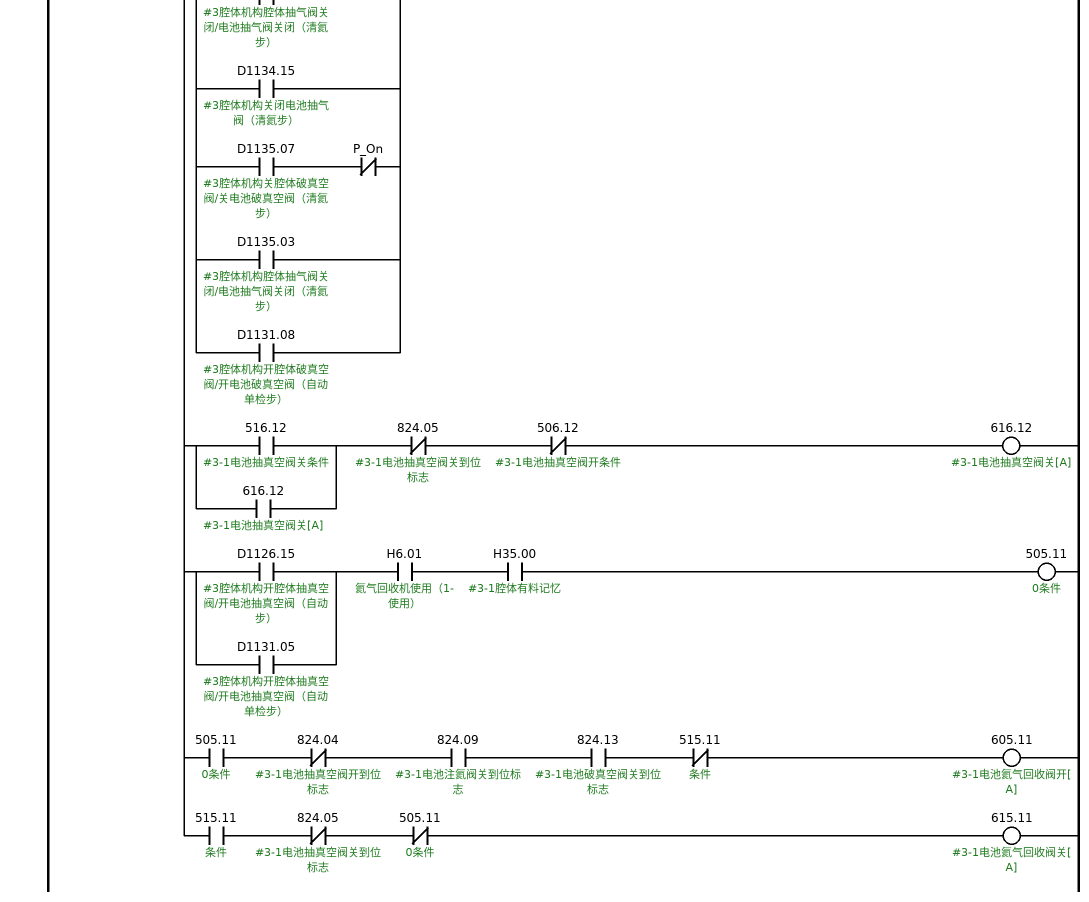
; rung 38: #3-1电池抽真空阀打开/关闭（A）
LD D1123.00  ; #3腔体机构单步/自动循环运行中（总）
OUT TR0
LD D1126.05  ; #3腔体机构腔体抽气阀打开/延时开电池抽气阀（自动步）
OR D1130.04  ; #3腔体机构腔体抽气阀打开/延时开#3-1电池抽气阀（自动单检步）
AND T2128  ; #3-1电池预抽压力正常判定延时（测试）
ANDNOT H36.00  ; #3-1电池泄漏
LD D1126.15  ; #3腔体机构开腔体抽真空阀/开电池抽真空阀（自动步）
OR D1131.05  ; #3腔体机构开腔体抽真空阀/开电池抽真空阀（自动单检步）
ANDNOT H6.01  ; 氦气回收机使用（1-使用）
ORLD
OR D1134.06  ; #3腔体机构腔体抽气阀打开/电池抽气阀打开（清氦步）
OR D1134.14  ; #3腔体机构腔体抽气阀打开/电池抽气阀打开（清氦步）
LD D1135.06  ; #3腔体机构开腔体破真空阀/开电池破真空阀/开腔体阀（清氦步）
ANDNOT P_On
ORLD
ANDLD
AND H35.00  ; #3-1腔体有料记忆
OUT 506.12  ; #3-1电池抽真空阀开条件
LD TR0
LD 506.12  ; #3-1电池抽真空阀开条件
OR 606.12  ; #3-1电池抽真空阀开[A]
ANDLD
ANDNOT 824.04  ; #3-1电池抽真空阀开到位标志
AND 824.09  ; #3-1电池注氦阀关到位标志
AND 824.13  ; #3-1电池破真空阀关到位标志
ANDNOT 516.12  ; #3-1电池抽真空阀关条件
OUT 606.12  ; #3-1电池抽真空阀开[A]
LD TR0
LD D1126.06  ; #3腔体机构关电池抽气阀（自动步）
OR D1127.00  ; #3腔体机构关腔体抽真空阀/关电池抽真空阀/开腔体阀（自动步）
OR D1130.05  ; #3腔体机构关#3-1电池抽气阀（自动单检步）
OR D1130.10  ; #3腔体机构关腔体氦检阀/关腔体抽气阀/关#3-1电池抽气阀（自动单检步）
OR D1131.06  ; #3腔体机构关腔体抽真空阀/关电池抽真空阀（自动单检步）
OR D1134.07  ; #3腔体机构腔体抽气阀关闭/电池抽气阀关闭（清氦步）
OR D1134.15  ; #3腔体机构关闭电池抽气阀（清氦步）
LD D1135.07  ; #3腔体机构关腔体破真空阀/关电池破真空阀（清氦步）
ANDNOT P_On
ORLD
OR D1135.03  ; #3腔体机构腔体抽气阀关闭/电池抽气阀关闭（清氦步）
OR D1131.08  ; #3腔体机构开腔体破真空阀/开电池破真空阀（自动单检步）
ANDLD
OUT 516.12  ; #3-1电池抽真空阀关条件
OUT 515.11  ; 条件
LD TR0
LD 516.12  ; #3-1电池抽真空阀关条件
OR 616.12  ; #3-1电池抽真空阀关[A]
ANDLD
ANDNOT 824.05  ; #3-1电池抽真空阀关到位标志
ANDNOT 506.12  ; #3-1电池抽真空阀开条件
OUT 616.12  ; #3-1电池抽真空阀关[A]
LD TR0
LD D1126.15  ; #3腔体机构开腔体抽真空阀/开电池抽真空阀（自动步）
OR D1131.05  ; #3腔体机构开腔体抽真空阀/开电池抽真空阀（自动单检步）
ANDLD
AND H6.01  ; 氦气回收机使用（1-使用）
AND H35.00  ; #3-1腔体有料记忆
OUT 505.11  ; 0条件
LD TR0
AND 505.11  ; 0条件
ANDNOT 824.04  ; #3-1电池抽真空阀开到位标志
AND 824.09  ; #3-1电池注氦阀关到位标志
AND 824.13  ; #3-1电池破真空阀关到位标志
ANDNOT 515.11  ; 条件
OUT 605.11  ; #3-1电池氦气回收阀开[A]
LD TR0
AND 515.11  ; 条件
ANDNOT 824.05  ; #3-1电池抽真空阀关到位标志
ANDNOT 505.11  ; 0条件
OUT 615.11  ; #3-1电池氦气回收阀关[A]

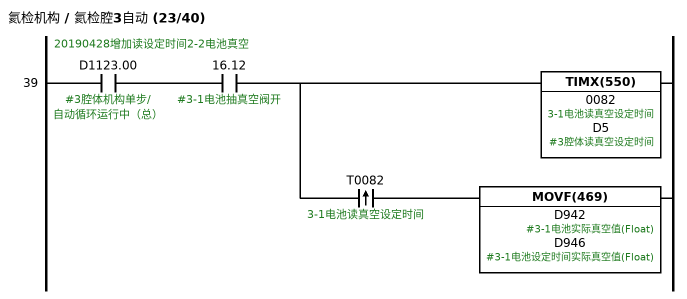
; rung 39: 20190428增加读设定时间2-2电池真空
LD D1123.00  ; #3腔体机构单步/自动循环运行中（总）
AND 16.12  ; #3-1电池抽真空阀开
TIMX(550) 0082 D5  ; #3腔体读真空设定时间, 3-1电池读真空设定时间
@AND T0082  ; 3-1电池读真空设定时间
MOVF(469) D942 D946  ; #3-1电池实际真空值(Float), #3-1电池设定时间实际真空值(Float)

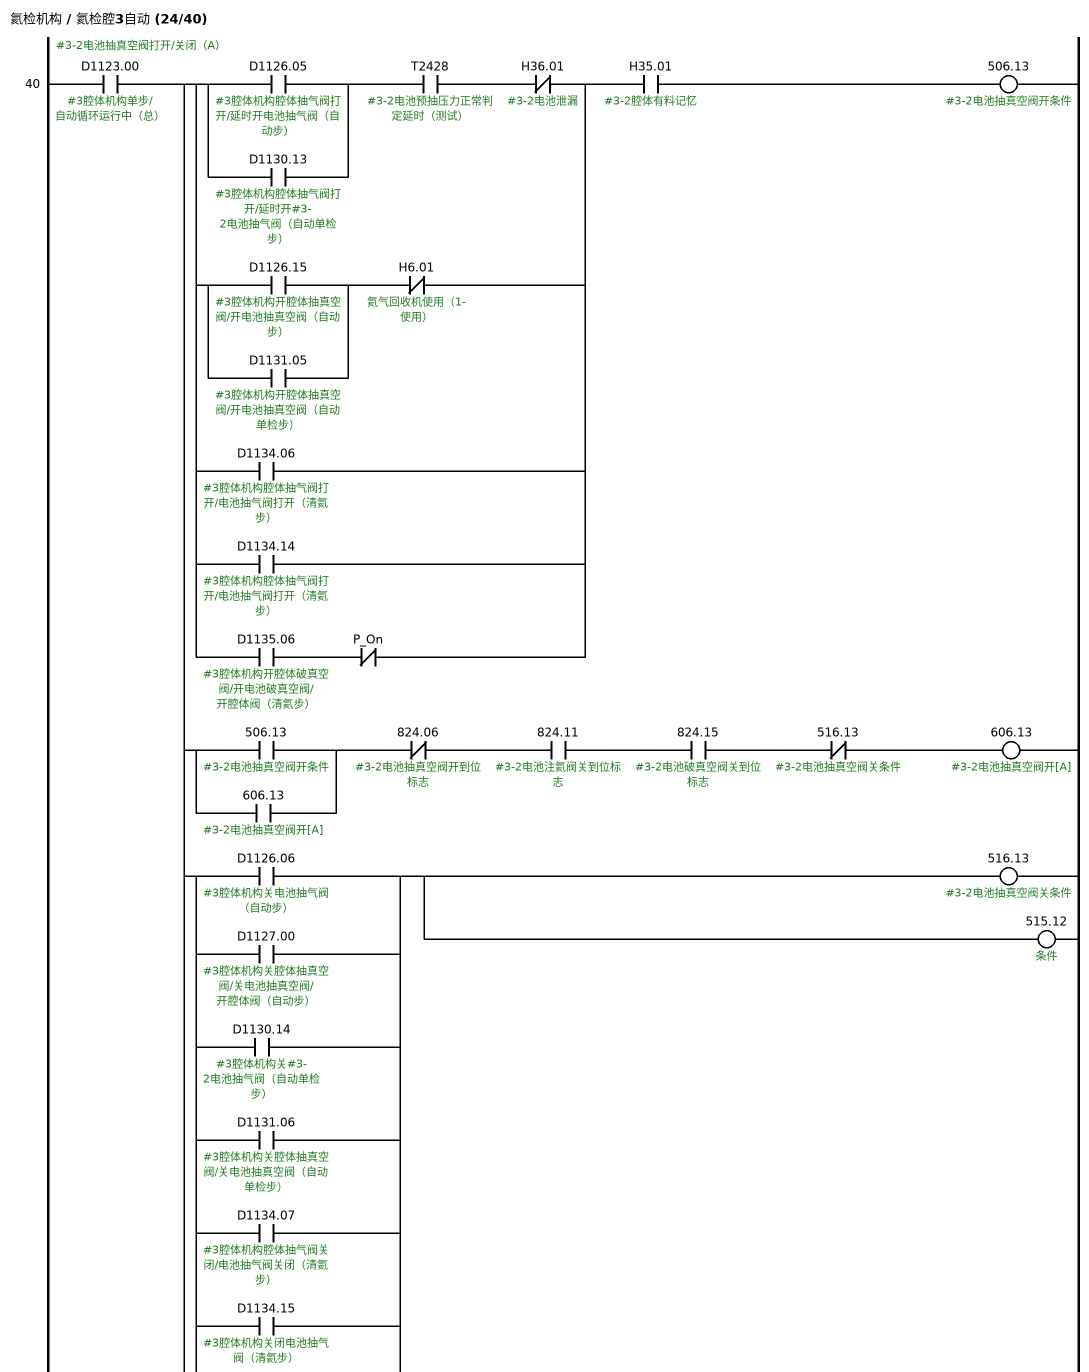

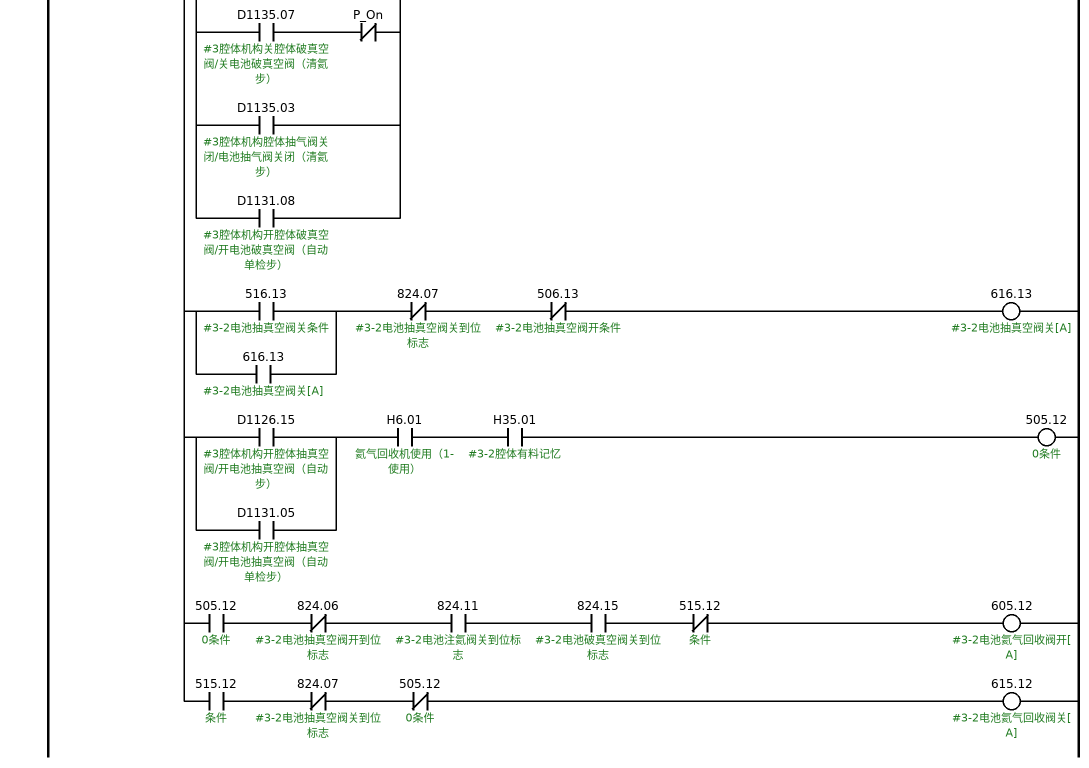
; rung 40: #3-2电池抽真空阀打开/关闭（A）
LD D1123.00  ; #3腔体机构单步/自动循环运行中（总）
OUT TR0
LD D1126.05  ; #3腔体机构腔体抽气阀打开/延时开电池抽气阀（自动步）
OR D1130.13  ; #3腔体机构腔体抽气阀打开/延时开#3-2电池抽气阀（自动单检步）
AND T2428  ; #3-2电池预抽压力正常判定延时（测试）
ANDNOT H36.01  ; #3-2电池泄漏
LD D1126.15  ; #3腔体机构开腔体抽真空阀/开电池抽真空阀（自动步）
OR D1131.05  ; #3腔体机构开腔体抽真空阀/开电池抽真空阀（自动单检步）
ANDNOT H6.01  ; 氦气回收机使用（1-使用）
ORLD
OR D1134.06  ; #3腔体机构腔体抽气阀打开/电池抽气阀打开（清氦步）
OR D1134.14  ; #3腔体机构腔体抽气阀打开/电池抽气阀打开（清氦步）
LD D1135.06  ; #3腔体机构开腔体破真空阀/开电池破真空阀/开腔体阀（清氦步）
ANDNOT P_On
ORLD
ANDLD
AND H35.01  ; #3-2腔体有料记忆
OUT 506.13  ; #3-2电池抽真空阀开条件
LD TR0
LD 506.13  ; #3-2电池抽真空阀开条件
OR 606.13  ; #3-2电池抽真空阀开[A]
ANDLD
ANDNOT 824.06  ; #3-2电池抽真空阀开到位标志
AND 824.11  ; #3-2电池注氦阀关到位标志
AND 824.15  ; #3-2电池破真空阀关到位标志
ANDNOT 516.13  ; #3-2电池抽真空阀关条件
OUT 606.13  ; #3-2电池抽真空阀开[A]
LD TR0
LD D1126.06  ; #3腔体机构关电池抽气阀（自动步）
OR D1127.00  ; #3腔体机构关腔体抽真空阀/关电池抽真空阀/开腔体阀（自动步）
OR D1130.14  ; #3腔体机构关#3-2电池抽气阀（自动单检步）
OR D1131.06  ; #3腔体机构关腔体抽真空阀/关电池抽真空阀（自动单检步）
OR D1134.07  ; #3腔体机构腔体抽气阀关闭/电池抽气阀关闭（清氦步）
OR D1134.15  ; #3腔体机构关闭电池抽气阀（清氦步）
LD D1135.07  ; #3腔体机构关腔体破真空阀/关电池破真空阀（清氦步）
ANDNOT P_On
ORLD
OR D1135.03  ; #3腔体机构腔体抽气阀关闭/电池抽气阀关闭（清氦步）
OR D1131.08  ; #3腔体机构开腔体破真空阀/开电池破真空阀（自动单检步）
ANDLD
OUT 516.13  ; #3-2电池抽真空阀关条件
OUT 515.12  ; 条件
LD TR0
LD 516.13  ; #3-2电池抽真空阀关条件
OR 616.13  ; #3-2电池抽真空阀关[A]
ANDLD
ANDNOT 824.07  ; #3-2电池抽真空阀关到位标志
ANDNOT 506.13  ; #3-2电池抽真空阀开条件
OUT 616.13  ; #3-2电池抽真空阀关[A]
LD TR0
LD D1126.15  ; #3腔体机构开腔体抽真空阀/开电池抽真空阀（自动步）
OR D1131.05  ; #3腔体机构开腔体抽真空阀/开电池抽真空阀（自动单检步）
ANDLD
AND H6.01  ; 氦气回收机使用（1-使用）
AND H35.01  ; #3-2腔体有料记忆
OUT 505.12  ; 0条件
LD TR0
AND 505.12  ; 0条件
ANDNOT 824.06  ; #3-2电池抽真空阀开到位标志
AND 824.11  ; #3-2电池注氦阀关到位标志
AND 824.15  ; #3-2电池破真空阀关到位标志
ANDNOT 515.12  ; 条件
OUT 605.12  ; #3-2电池氦气回收阀开[A]
LD TR0
AND 515.12  ; 条件
ANDNOT 824.07  ; #3-2电池抽真空阀关到位标志
ANDNOT 505.12  ; 0条件
OUT 615.12  ; #3-2电池氦气回收阀关[A]

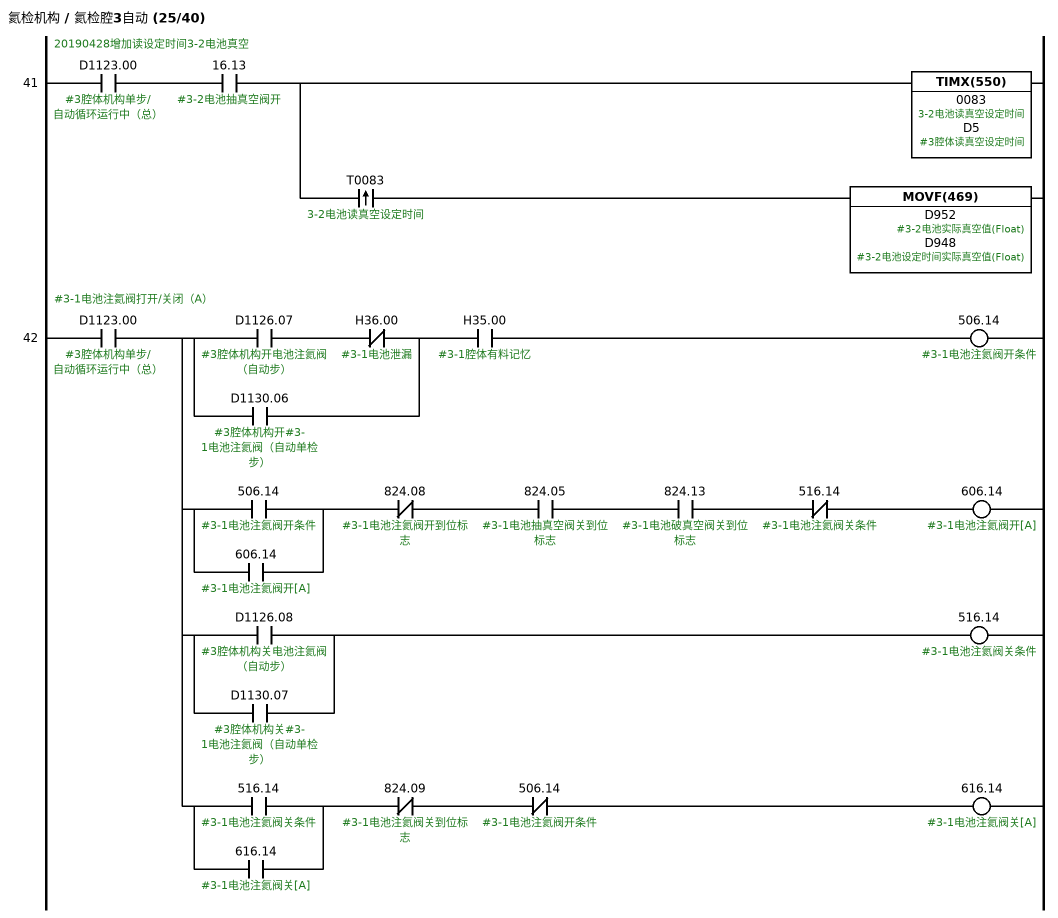
; rung 41: 20190428增加读设定时间3-2电池真空
LD D1123.00  ; #3腔体机构单步/自动循环运行中（总）
AND 16.13  ; #3-2电池抽真空阀开
TIMX(550) 0083 D5  ; #3腔体读真空设定时间, 3-2电池读真空设定时间
@AND T0083  ; 3-2电池读真空设定时间
MOVF(469) D952 D948  ; #3-2电池实际真空值(Float), #3-2电池设定时间实际真空值(Float)
; rung 42: #3-1电池注氦阀打开/关闭（A）
LD D1123.00  ; #3腔体机构单步/自动循环运行中（总）
OUT TR0
LD D1126.07  ; #3腔体机构开电池注氦阀（自动步）
ANDNOT H36.00  ; #3-1电池泄漏
OR D1130.06  ; #3腔体机构开#3-1电池注氦阀（自动单检步）
ANDLD
AND H35.00  ; #3-1腔体有料记忆
OUT 506.14  ; #3-1电池注氦阀开条件
LD TR0
LD 506.14  ; #3-1电池注氦阀开条件
OR 606.14  ; #3-1电池注氦阀开[A]
ANDLD
ANDNOT 824.08  ; #3-1电池注氦阀开到位标志
AND 824.05  ; #3-1电池抽真空阀关到位标志
AND 824.13  ; #3-1电池破真空阀关到位标志
ANDNOT 516.14  ; #3-1电池注氦阀关条件
OUT 606.14  ; #3-1电池注氦阀开[A]
LD TR0
LD D1126.08  ; #3腔体机构关电池注氦阀（自动步）
OR D1130.07  ; #3腔体机构关#3-1电池注氦阀（自动单检步）
ANDLD
OUT 516.14  ; #3-1电池注氦阀关条件
LD TR0
LD 516.14  ; #3-1电池注氦阀关条件
OR 616.14  ; #3-1电池注氦阀关[A]
ANDLD
ANDNOT 824.09  ; #3-1电池注氦阀关到位标志
ANDNOT 506.14  ; #3-1电池注氦阀开条件
OUT 616.14  ; #3-1电池注氦阀关[A]

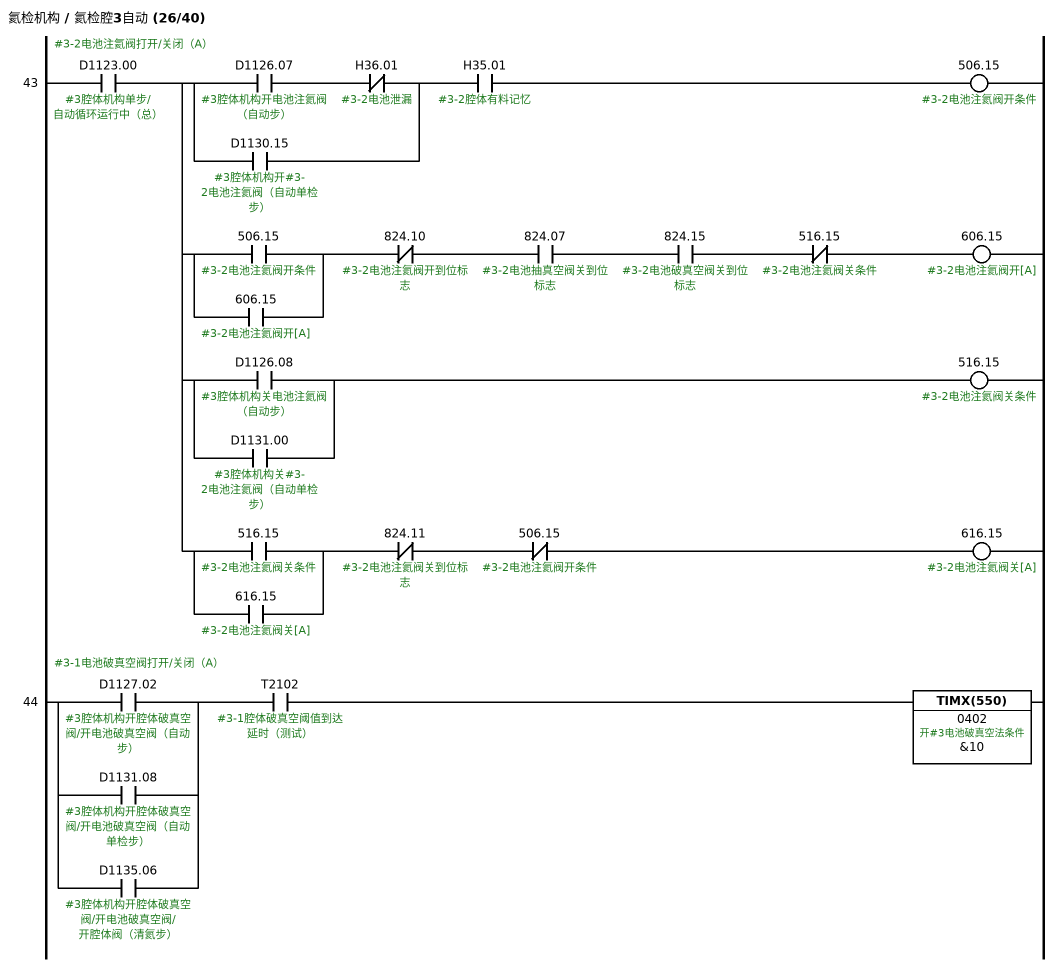
; rung 43: #3-2电池注氦阀打开/关闭（A）
LD D1123.00  ; #3腔体机构单步/自动循环运行中（总）
OUT TR0
LD D1126.07  ; #3腔体机构开电池注氦阀（自动步）
ANDNOT H36.01  ; #3-2电池泄漏
OR D1130.15  ; #3腔体机构开#3-2电池注氦阀（自动单检步）
ANDLD
AND H35.01  ; #3-2腔体有料记忆
OUT 506.15  ; #3-2电池注氦阀开条件
LD TR0
LD 506.15  ; #3-2电池注氦阀开条件
OR 606.15  ; #3-2电池注氦阀开[A]
ANDLD
ANDNOT 824.10  ; #3-2电池注氦阀开到位标志
AND 824.07  ; #3-2电池抽真空阀关到位标志
AND 824.15  ; #3-2电池破真空阀关到位标志
ANDNOT 516.15  ; #3-2电池注氦阀关条件
OUT 606.15  ; #3-2电池注氦阀开[A]
LD TR0
LD D1126.08  ; #3腔体机构关电池注氦阀（自动步）
OR D1131.00  ; #3腔体机构关#3-2电池注氦阀（自动单检步）
ANDLD
OUT 516.15  ; #3-2电池注氦阀关条件
LD TR0
LD 516.15  ; #3-2电池注氦阀关条件
OR 616.15  ; #3-2电池注氦阀关[A]
ANDLD
ANDNOT 824.11  ; #3-2电池注氦阀关到位标志
ANDNOT 506.15  ; #3-2电池注氦阀开条件
OUT 616.15  ; #3-2电池注氦阀关[A]
; rung 44: #3-1电池破真空阀打开/关闭（A）
LD D1127.02  ; #3腔体机构开腔体破真空阀/开电池破真空阀（自动步）
OR D1131.08  ; #3腔体机构开腔体破真空阀/开电池破真空阀（自动单检步）
OR D1135.06  ; #3腔体机构开腔体破真空阀/开电池破真空阀/开腔体阀（清氦步）
AND T2102  ; #3-1腔体破真空阈值到达延时（测试）
TIMX(550) 0402 &10  ; 开#3电池破真空法条件

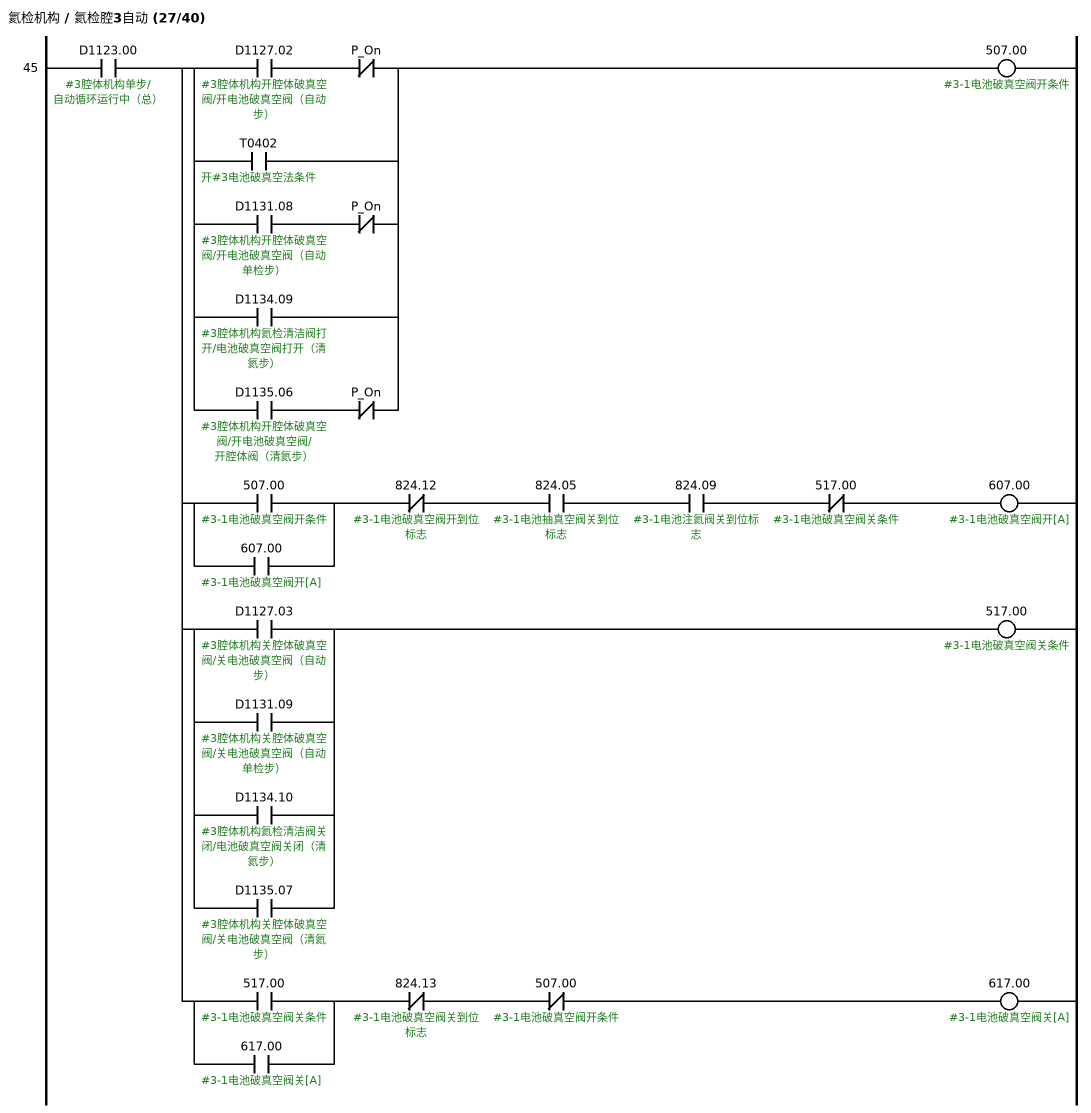
; rung 45
LD D1123.00  ; #3腔体机构单步/自动循环运行中（总）
OUT TR0
LD D1127.02  ; #3腔体机构开腔体破真空阀/开电池破真空阀（自动步）
ANDNOT P_On
OR T0402  ; 开#3电池破真空法条件
LD D1131.08  ; #3腔体机构开腔体破真空阀/开电池破真空阀（自动单检步）
ANDNOT P_On
ORLD
OR D1134.09  ; #3腔体机构氦检清洁阀打开/电池破真空阀打开（清氦步）
LD D1135.06  ; #3腔体机构开腔体破真空阀/开电池破真空阀/开腔体阀（清氦步）
ANDNOT P_On
ORLD
ANDLD
OUT 507.00  ; #3-1电池破真空阀开条件
LD TR0
LD 507.00  ; #3-1电池破真空阀开条件
OR 607.00  ; #3-1电池破真空阀开[A]
ANDLD
ANDNOT 824.12  ; #3-1电池破真空阀开到位标志
AND 824.05  ; #3-1电池抽真空阀关到位标志
AND 824.09  ; #3-1电池注氦阀关到位标志
ANDNOT 517.00  ; #3-1电池破真空阀关条件
OUT 607.00  ; #3-1电池破真空阀开[A]
LD TR0
LD D1127.03  ; #3腔体机构关腔体破真空阀/关电池破真空阀（自动步）
OR D1131.09  ; #3腔体机构关腔体破真空阀/关电池破真空阀（自动单检步）
OR D1134.10  ; #3腔体机构氦检清洁阀关闭/电池破真空阀关闭（清氦步）
OR D1135.07  ; #3腔体机构关腔体破真空阀/关电池破真空阀（清氦步）
ANDLD
OUT 517.00  ; #3-1电池破真空阀关条件
LD TR0
LD 517.00  ; #3-1电池破真空阀关条件
OR 617.00  ; #3-1电池破真空阀关[A]
ANDLD
ANDNOT 824.13  ; #3-1电池破真空阀关到位标志
ANDNOT 507.00  ; #3-1电池破真空阀开条件
OUT 617.00  ; #3-1电池破真空阀关[A]

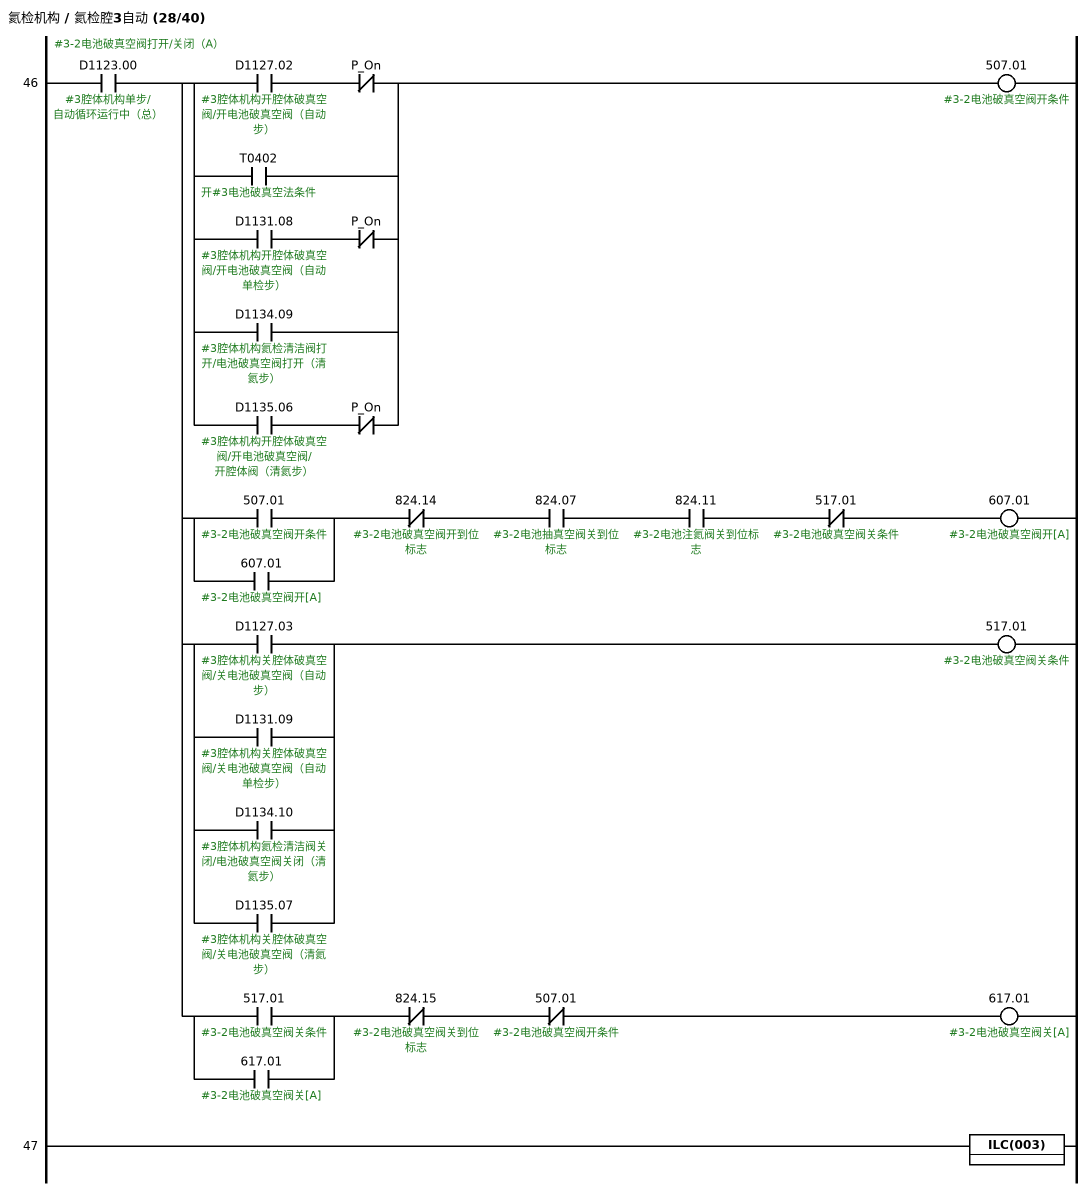
; rung 46: #3-2电池破真空阀打开/关闭（A）
LD D1123.00  ; #3腔体机构单步/自动循环运行中（总）
OUT TR0
LD D1127.02  ; #3腔体机构开腔体破真空阀/开电池破真空阀（自动步）
ANDNOT P_On
OR T0402  ; 开#3电池破真空法条件
LD D1131.08  ; #3腔体机构开腔体破真空阀/开电池破真空阀（自动单检步）
ANDNOT P_On
ORLD
OR D1134.09  ; #3腔体机构氦检清洁阀打开/电池破真空阀打开（清氦步）
LD D1135.06  ; #3腔体机构开腔体破真空阀/开电池破真空阀/开腔体阀（清氦步）
ANDNOT P_On
ORLD
ANDLD
OUT 507.01  ; #3-2电池破真空阀开条件
LD TR0
LD 507.01  ; #3-2电池破真空阀开条件
OR 607.01  ; #3-2电池破真空阀开[A]
ANDLD
ANDNOT 824.14  ; #3-2电池破真空阀开到位标志
AND 824.07  ; #3-2电池抽真空阀关到位标志
AND 824.11  ; #3-2电池注氦阀关到位标志
ANDNOT 517.01  ; #3-2电池破真空阀关条件
OUT 607.01  ; #3-2电池破真空阀开[A]
LD TR0
LD D1127.03  ; #3腔体机构关腔体破真空阀/关电池破真空阀（自动步）
OR D1131.09  ; #3腔体机构关腔体破真空阀/关电池破真空阀（自动单检步）
OR D1134.10  ; #3腔体机构氦检清洁阀关闭/电池破真空阀关闭（清氦步）
OR D1135.07  ; #3腔体机构关腔体破真空阀/关电池破真空阀（清氦步）
ANDLD
OUT 517.01  ; #3-2电池破真空阀关条件
LD TR0
LD 517.01  ; #3-2电池破真空阀关条件
OR 617.01  ; #3-2电池破真空阀关[A]
ANDLD
ANDNOT 824.15  ; #3-2电池破真空阀关到位标志
ANDNOT 507.01  ; #3-2电池破真空阀开条件
OUT 617.01  ; #3-2电池破真空阀关[A]
; rung 47
ILC(003)

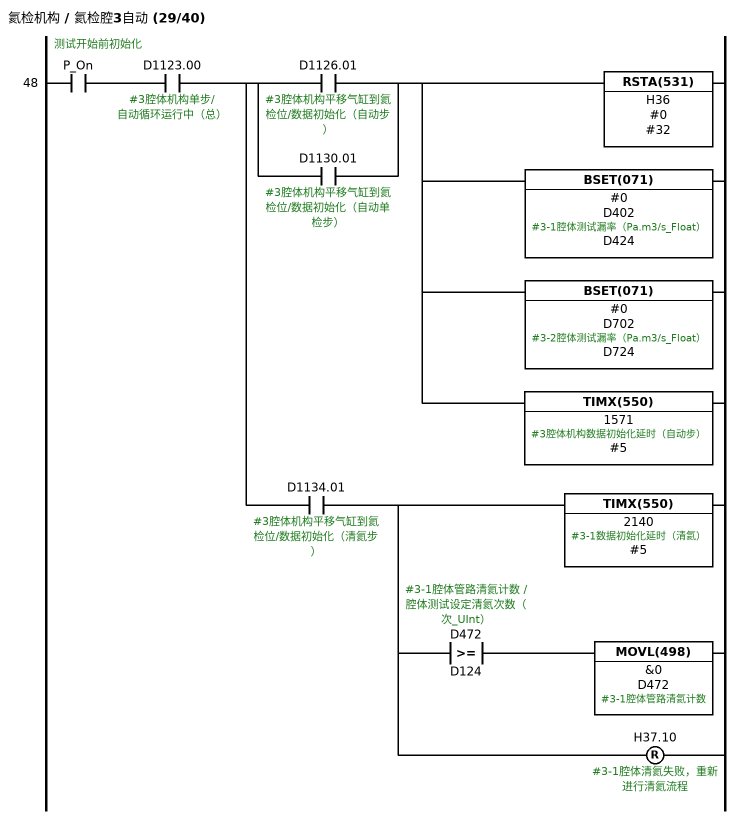
; rung 48: 测试开始前初始化
LD P_On
AND D1123.00  ; #3腔体机构单步/自动循环运行中（总）
OUT TR0
LD D1126.01  ; #3腔体机构平移气缸到氦检位/数据初始化（自动步）
OR D1130.01  ; #3腔体机构平移气缸到氦检位/数据初始化（自动单检步）
ANDLD
RSTA(531) H36 #0 #32
BSET(071) #0 D402 D424  ; #3-1腔体测试漏率（Pa.m3/s_Float）
BSET(071) #0 D702 D724  ; #3-2腔体测试漏率（Pa.m3/s_Float）
TIMX(550) 1571 #5  ; #3腔体机构数据初始化延时（自动步）
LD TR0
AND D1134.01  ; #3腔体机构平移气缸到氦检位/数据初始化（清氦步）
OUT TR0
TIMX(550) 2140 #5  ; #3-1数据初始化延时（清氦）
AND>=(325) D472 D124  ; #3-1腔体管路清氦计数, 腔体测试设定清氦次数（次_UInt）
MOVL(498) &0 D472  ; #3-1腔体管路清氦计数
LD TR0
RSET H37.10  ; #3-1腔体清氦失败，重新进行清氦流程

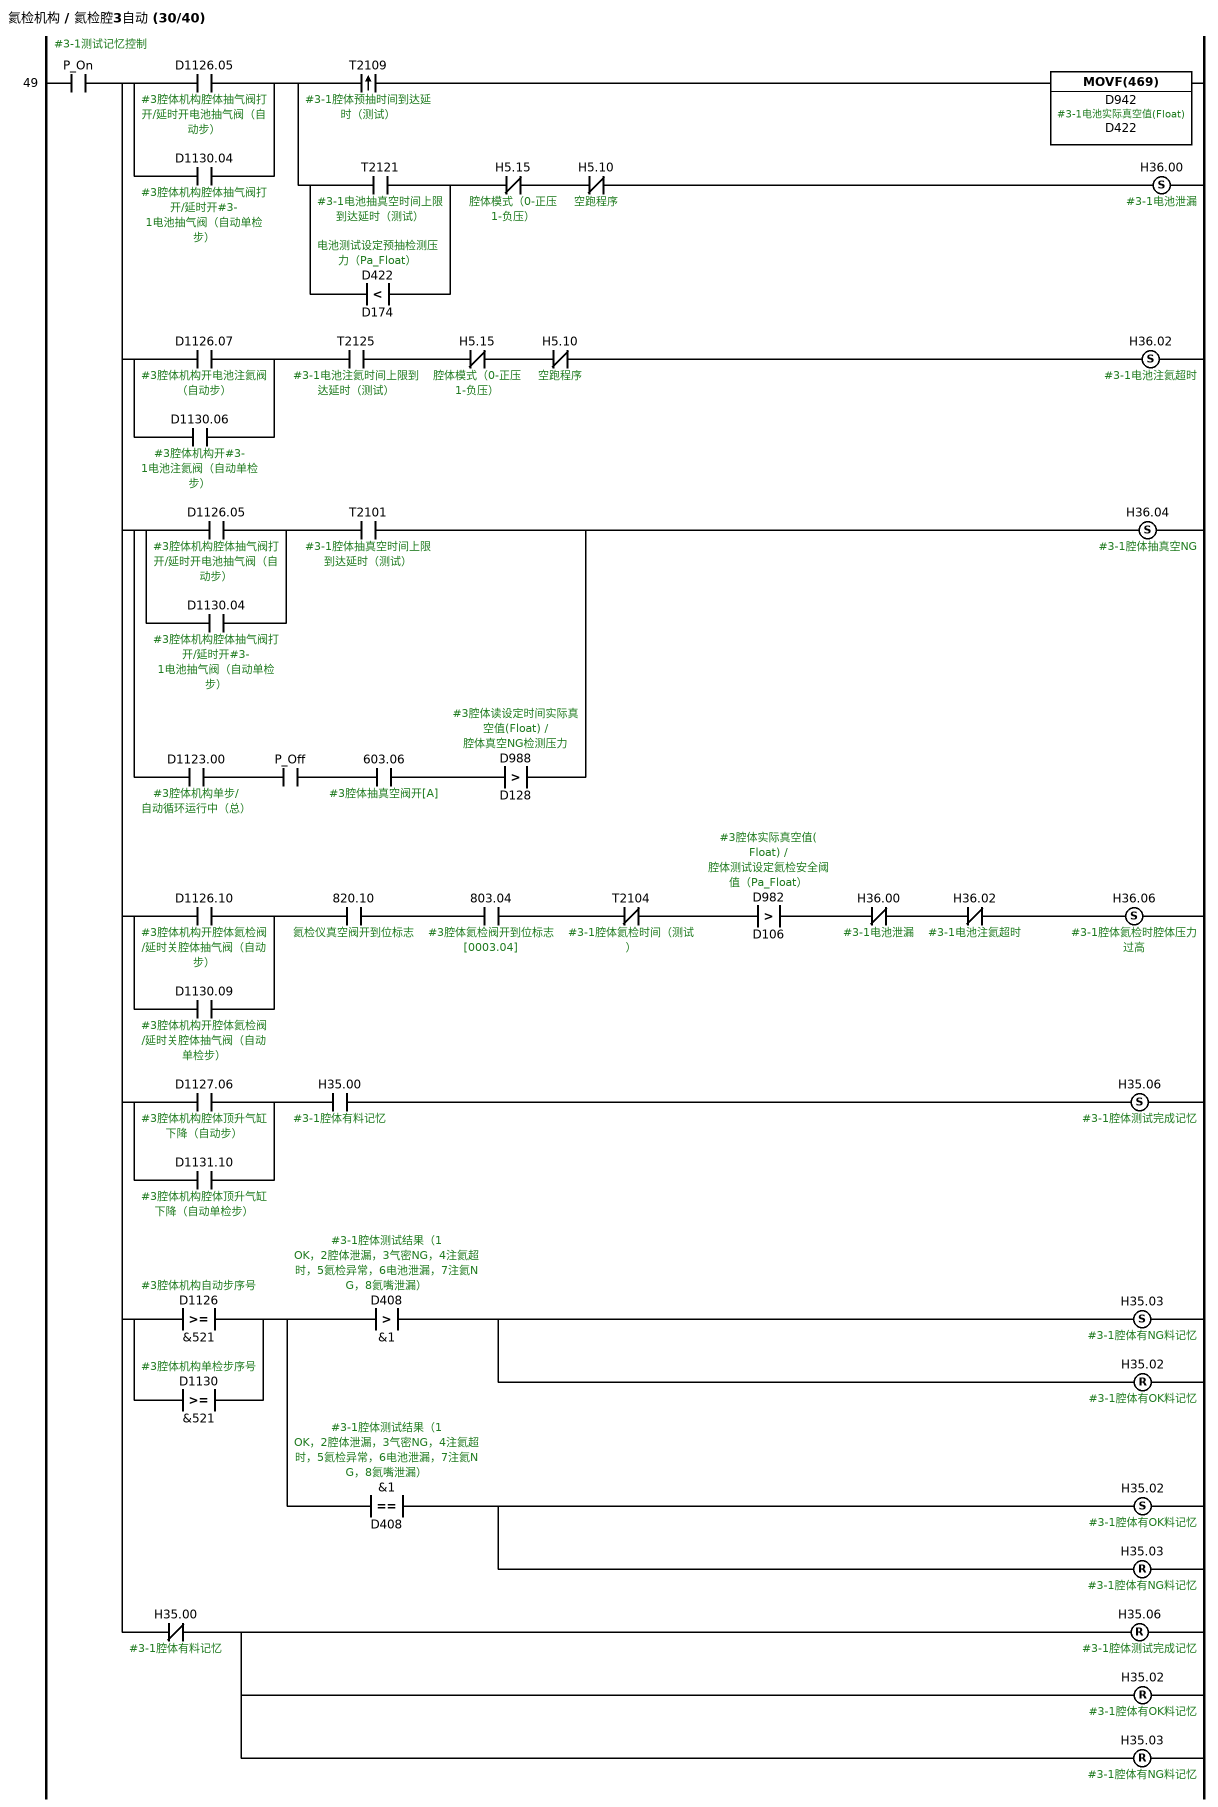
; rung 49: #3-1测试记忆控制
LD P_On
OUT TR0
LD D1126.05  ; #3腔体机构腔体抽气阀打开/延时开电池抽气阀（自动步）
OR D1130.04  ; #3腔体机构腔体抽气阀打开/延时开#3-1电池抽气阀（自动单检步）
ANDLD
OUT TR1
@AND T2109  ; #3-1腔体预抽时间到达延时（测试）
MOVF(469) D942 D422  ; #3-1电池实际真空值(Float)
LD TR1
LD T2121  ; #3-1电池抽真空时间上限到达延时（测试）
OR<F(331) D422 D174  ; 电池测试设定预抽检测压力（Pa_Float）
ANDLD
ANDNOT H5.15  ; 腔体模式（0-正压 1-负压）
ANDNOT H5.10  ; 空跑程序
SET H36.00  ; #3-1电池泄漏
LD TR0
LD D1126.07  ; #3腔体机构开电池注氦阀（自动步）
OR D1130.06  ; #3腔体机构开#3-1电池注氦阀（自动单检步）
ANDLD
AND T2125  ; #3-1电池注氦时间上限到达延时（测试）
ANDNOT H5.15  ; 腔体模式（0-正压 1-负压）
ANDNOT H5.10  ; 空跑程序
SET H36.02  ; #3-1电池注氦超时
LD TR0
LD D1126.05  ; #3腔体机构腔体抽气阀打开/延时开电池抽气阀（自动步）
OR D1130.04  ; #3腔体机构腔体抽气阀打开/延时开#3-1电池抽气阀（自动单检步）
AND T2101  ; #3-1腔体抽真空时间上限到达延时（测试）
LD D1123.00  ; #3腔体机构单步/自动循环运行中（总）
AND P_Off
AND 603.06  ; #3腔体抽真空阀开[A]
AND>F(333) D988 D128  ; #3腔体读设定时间实际真空值(Float), 腔体真空NG检测压力
ORLD
ANDLD
SET H36.04  ; #3-1腔体抽真空NG
LD TR0
LD D1126.10  ; #3腔体机构开腔体氦检阀/延时关腔体抽气阀（自动步）
OR D1130.09  ; #3腔体机构开腔体氦检阀/延时关腔体抽气阀（自动单检步）
ANDLD
AND 820.10  ; 氦检仪真空阀开到位标志
AND 803.04  ; #3腔体氦检阀开到位标志[0003.04]
ANDNOT T2104  ; #3-1腔体氦检时间（测试）
AND>F(333) D982 D106  ; #3腔体实际真空值(Float), 腔体测试设定氦检安全阈值（Pa_Float）
ANDNOT H36.00  ; #3-1电池泄漏
ANDNOT H36.02  ; #3-1电池注氦超时
SET H36.06  ; #3-1腔体氦检时腔体压力过高
LD TR0
LD D1127.06  ; #3腔体机构腔体顶升气缸下降（自动步）
OR D1131.10  ; #3腔体机构腔体顶升气缸下降（自动单检步）
ANDLD
AND H35.00  ; #3-1腔体有料记忆
SET H35.06  ; #3-1腔体测试完成记忆
LD TR0
LD>=L(326) D1126 &521  ; #3腔体机构自动步序号
OR>=L(326) D1130 &521  ; #3腔体机构单检步序号
ANDLD
OUT TR1
AND>(320) D408 &1  ; #3-1腔体测试结果（1 OK，2腔体泄漏，3气密NG，4注氦超时，5氦检异常，6电池泄漏，7注氦NG，8氦嘴泄漏）
SET H35.03  ; #3-1腔体有NG料记忆
RSET H35.02  ; #3-1腔体有OK料记忆
LD TR1
AND=(300) &1 D408  ; #3-1腔体测试结果（1 OK，2腔体泄漏，3气密NG，4注氦超时，5氦检异常，6电池泄漏，7注氦NG，8氦嘴泄漏）
SET H35.02  ; #3-1腔体有OK料记忆
RSET H35.03  ; #3-1腔体有NG料记忆
LD TR0
ANDNOT H35.00  ; #3-1腔体有料记忆
RSET H35.06  ; #3-1腔体测试完成记忆
RSET H35.02  ; #3-1腔体有OK料记忆
RSET H35.03  ; #3-1腔体有NG料记忆

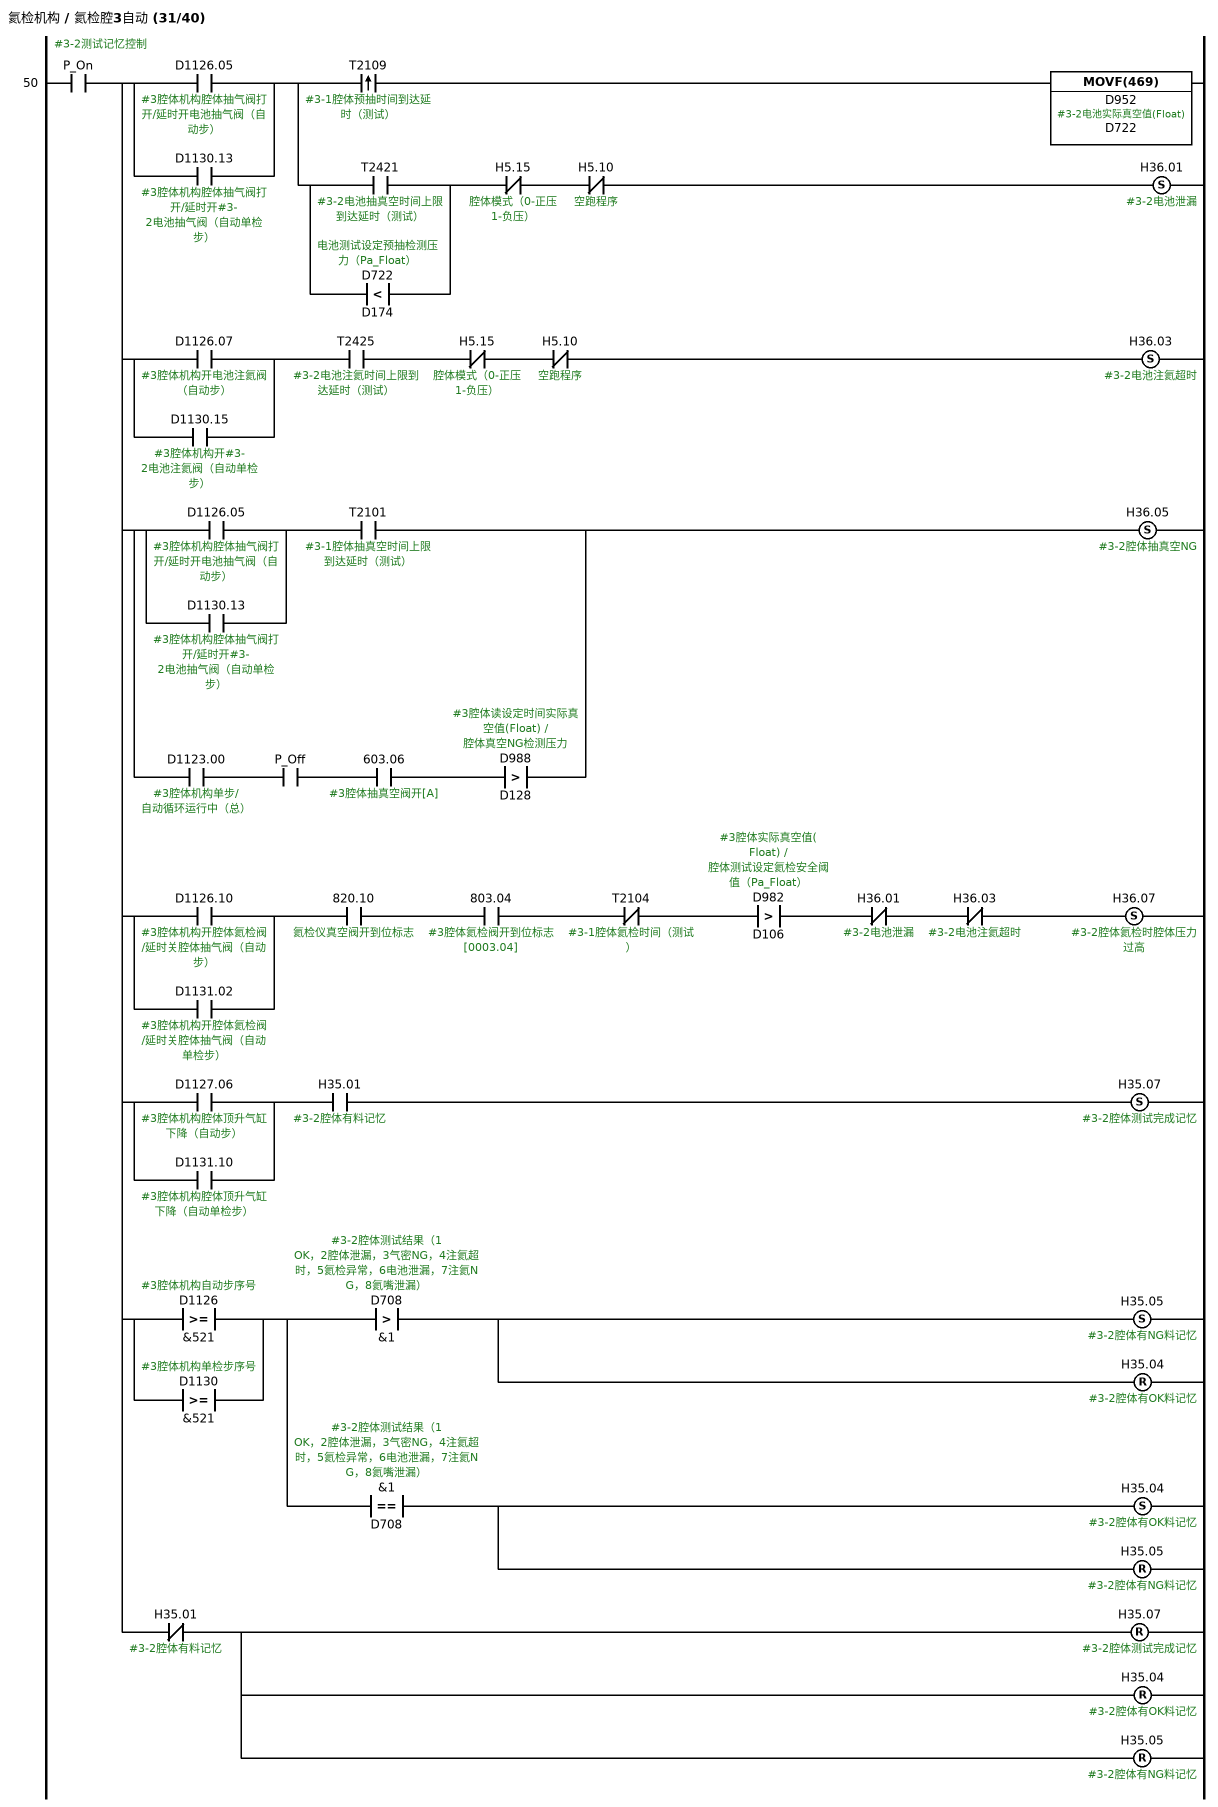
; rung 50: #3-2测试记忆控制
LD P_On
OUT TR0
LD D1126.05  ; #3腔体机构腔体抽气阀打开/延时开电池抽气阀（自动步）
OR D1130.13  ; #3腔体机构腔体抽气阀打开/延时开#3-2电池抽气阀（自动单检步）
ANDLD
OUT TR1
@AND T2109  ; #3-1腔体预抽时间到达延时（测试）
MOVF(469) D952 D722  ; #3-2电池实际真空值(Float)
LD TR1
LD T2421  ; #3-2电池抽真空时间上限到达延时（测试）
OR<F(331) D722 D174  ; 电池测试设定预抽检测压力（Pa_Float）
ANDLD
ANDNOT H5.15  ; 腔体模式（0-正压 1-负压）
ANDNOT H5.10  ; 空跑程序
SET H36.01  ; #3-2电池泄漏
LD TR0
LD D1126.07  ; #3腔体机构开电池注氦阀（自动步）
OR D1130.15  ; #3腔体机构开#3-2电池注氦阀（自动单检步）
ANDLD
AND T2425  ; #3-2电池注氦时间上限到达延时（测试）
ANDNOT H5.15  ; 腔体模式（0-正压 1-负压）
ANDNOT H5.10  ; 空跑程序
SET H36.03  ; #3-2电池注氦超时
LD TR0
LD D1126.05  ; #3腔体机构腔体抽气阀打开/延时开电池抽气阀（自动步）
OR D1130.13  ; #3腔体机构腔体抽气阀打开/延时开#3-2电池抽气阀（自动单检步）
AND T2101  ; #3-1腔体抽真空时间上限到达延时（测试）
LD D1123.00  ; #3腔体机构单步/自动循环运行中（总）
AND P_Off
AND 603.06  ; #3腔体抽真空阀开[A]
AND>F(333) D988 D128  ; #3腔体读设定时间实际真空值(Float), 腔体真空NG检测压力
ORLD
ANDLD
SET H36.05  ; #3-2腔体抽真空NG
LD TR0
LD D1126.10  ; #3腔体机构开腔体氦检阀/延时关腔体抽气阀（自动步）
OR D1131.02  ; #3腔体机构开腔体氦检阀/延时关腔体抽气阀（自动单检步）
ANDLD
AND 820.10  ; 氦检仪真空阀开到位标志
AND 803.04  ; #3腔体氦检阀开到位标志[0003.04]
ANDNOT T2104  ; #3-1腔体氦检时间（测试）
AND>F(333) D982 D106  ; #3腔体实际真空值(Float), 腔体测试设定氦检安全阈值（Pa_Float）
ANDNOT H36.01  ; #3-2电池泄漏
ANDNOT H36.03  ; #3-2电池注氦超时
SET H36.07  ; #3-2腔体氦检时腔体压力过高
LD TR0
LD D1127.06  ; #3腔体机构腔体顶升气缸下降（自动步）
OR D1131.10  ; #3腔体机构腔体顶升气缸下降（自动单检步）
ANDLD
AND H35.01  ; #3-2腔体有料记忆
SET H35.07  ; #3-2腔体测试完成记忆
LD TR0
LD>=L(326) D1126 &521  ; #3腔体机构自动步序号
OR>=L(326) D1130 &521  ; #3腔体机构单检步序号
ANDLD
OUT TR1
AND>(320) D708 &1  ; #3-2腔体测试结果（1 OK，2腔体泄漏，3气密NG，4注氦超时，5氦检异常，6电池泄漏，7注氦NG，8氦嘴泄漏）
SET H35.05  ; #3-2腔体有NG料记忆
RSET H35.04  ; #3-2腔体有OK料记忆
LD TR1
AND=(300) &1 D708  ; #3-2腔体测试结果（1 OK，2腔体泄漏，3气密NG，4注氦超时，5氦检异常，6电池泄漏，7注氦NG，8氦嘴泄漏）
SET H35.04  ; #3-2腔体有OK料记忆
RSET H35.05  ; #3-2腔体有NG料记忆
LD TR0
ANDNOT H35.01  ; #3-2腔体有料记忆
RSET H35.07  ; #3-2腔体测试完成记忆
RSET H35.04  ; #3-2腔体有OK料记忆
RSET H35.05  ; #3-2腔体有NG料记忆

